(* CODESYS project BaseHts.library
   Company: Vistaprint
   Version: 0.0.0.48
   Description: 0.0.0.48 - Add AutoMode to HRU
      
      0.0.0.47 - Some Bugs in DPJ fixed
      
      0.0.0.46 - BaseElements 0.0.1.18
      	Some Bugs in DPJ, JUN fixed
      
      0.0.0.45 - BaseElements 0.0.1.17
      	MTR/sta_RUN Bug fixed
      
      0.0.0.44 - New Libs BasePLC 0.3.4.8, BaseElements 0.0.1.16
      
      0.0.0.43 - DPJ reworked (Missed Shirt Problem)
      
      0.0.0.42 - MER - new parameter added
      	HFE reworked
      
      0.0.0.41 - BasePLC V0.3.4.5; BaseElements V0.0.1.9
      
      0.0.0.40 - Add MTR Parameter dinWaitBetweenSensorAndReservation_um
      
      0.0.0.39 - Bug fixed in HFE, CHD; FOC and FOD added
      
      0.0.0.34 - JUN / DPJ replaced with version from Shirtstream
      
      0.0.0.32 - HFE from Lvl1 to Lvl2 and reworked
      
      0.0.0.30 - BaseElements 0.0.1.5 BasePLC 0.3.4.3 included, Tc2_SerialCom
      
      0.0.0.29 - BaseElements 0.0.1.2 BasePLC 0.3.4.2 included; FB_CtrlModule moved to BaseElements
      
      0.0.0.28 - Added ADS data channel to FB_HPS
      for shirt request from Heatpress
      
      0.0.0.27 - Added bolStopReleaseHangers
      
      0.0.0.26 - DPJ.sta_RUN Entry action reworked
      
      0.0.0.25 - Error JUN changed
      
      0.0.0.24 - Rising Edge detection of bolBringShirt in HPS
      
      0.0.0.23 - HTS, hanger turned line wait at SEP
      
      0.0.0.22 - Bug fixed in STOPbusy
      
      0.0.0.21 - Bugs fixed in HPS
      
      0.0.0.20 - HPS with new Child SEP
      	New BaseElements 0.0.0.20
      
      0.0.0.19 - Alternativ status for run sequence added; Timing reworked in MER jam detection;
      DPJ STOPBusy reworked, HRU Errors reworked, DPJ new Errors 12 and 13 added
      
      0.0.0.18 - Timeout Run / Stop sequence added
      
      0.0.0.17 - EMO reworked in BaseCtrlModule; CHD "destination full" reworked; AddStpGrp, AddRunGrp removed
      
      0.0.0.16 - Back to BasePLC Lib. V3.3.5 beacuase of PageFaults
      
      0.0.0.15 - Rebuild
      
      0.0.0.14 - Bugzilla ID 03: BufferFull for LineControl added
      
      0.0.0.13 - Bugzilla ID 55: reworked refill of SLB/STB
      
      0.0.0.12 - Update of BasePLC 0.3.3.7, BaseElements 0.0.0.17
      
      0.0.0.11 - Add more controllers to the library (LAI, CHD, HFE, PLS, JUN, DPJ, MER, HRU, HPS, COS, STB, SLB)
      
      0.0.0.10 - Clear pending command to prevent automatic recovery in sta_STOPBusy
      
      0.0.0.9 - BugFix in sub state "cSTA_SUB_CHECK_GROUP_STATUS" from run and stop sequence. Insert new "bolChecked" flag to detect if the sequence has been processed correctly.
      
      0.0.0.8 - Add TSTOP in checkChildAlmClass
      
      0.0.0.7- General revision of behaviour in case of emergency off (state EOFF) and general error (state ERROR). New handling for module specific interface.
      
      0.0.0.6 - Go to EOFFBusy if not in sta_EOFF
      
      0.0.0.5 - In Always: go to EOFFBusy at generalFault
      
      0.0.0.4 - In Always: go to EOFFBusy not to EOFF at emergency stop
      
      0.0.0.3 - Remove CurrentItemCounter and his inputs
      
      0.0.0.2 - Changes after first use in simulation in ICL Module
      
      0.0.0.1 - First release
   Author: AVME/DSC
   Title: Base_Hts

Project tree, tasks and I/O mapping:
  libraries: Base_Elements, 0.0.1.18 (Vistaprint); Base_PLC, 0.3.4.8 (Vistaprint); Tc2_Standard, 3.3.0.0 (Beckhoff Automation GmbH); Tc2_System, 3.3.5.0 (Beckhoff Automation GmbH); Tc2_Utilities, 3.3.7.0 (Beckhoff Automation GmbH); Tc3_Module, 3.3.5.0 (Beckhoff Automation GmbH)
  POUs/
    Controller/
      Driver/
        FOD/
          Infrastructure/
            function block FB_DecodeCanRxMessage [ST]
            function block fb_GenerateCanTxMessage [ST]
          function block FB_ReceiveFolderState [ST]: init
          function block FB_SendFolderMessage [ST]: init
          data type T_FOD
          data type T_FOD_Cfg
          data type T_FOD_Cur
          data type T_FOD_StateMachine
      Lvl0/
        CHD (Cross Hanger Detection)/
          global variables CHD_CmdState
          global variables Const_CHD
          function block FB_CHD [ST]: Always, FB_init, getCmdState, getCtrlSIf, IoInBridge, IoOutBridge, sta_ERROR, sta_ERRORQuit, sta_OFF, sta_OFFBusy, sta_PON, sta_RUN, sta_RUNBusy, sta_STOP, sta_STOPBusy, StateMachine
          data type T_CheckElement
          data type T_Ctrl_SIf_CHD
          data type T_Ctrl_SIf_CHD_Cfg
          data type T_Ctrl_SIf_CHD_Cur
          data type T_Ctrl_SIf_CHD_In
          data type T_Ctrl_SIf_CHD_Out
          data type T_Ctrl_SIf_CHD_Par
        FOC (Folder Communication)/
          function block FB_FOC [ST]: Always, FB_init, getCmdState, getCtrlSIf, IoInBridge, IoOutBridge, sta_ERROR, sta_OFF, sta_RELEASE, sta_RUN, sta_RUNbusy, StateMachine
          global variables FOC_CmdState
          data type T_Ctrl_SIf_FOC
          data type T_Ctrl_SIf_FOC_Cfg
          data type T_Ctrl_SIf_FOC_Cur
          data type T_Ctrl_SIf_FOC_In
          data type T_Ctrl_SIf_FOC_Out
          data type T_Ctrl_SIf_FOC_Par
        HRU (Hanger Rotation Unit)/
          function block FB_HRU [ST]: Always, FB_init, getCmdState, getCtrlSIf, IoInBridge, IoOutBridge, sta_EJECT, sta_EJECTBusy, sta_OFF, sta_OFFBusy, sta_RETRACT, sta_RETRACTBusy, sta_ROTATE, sta_ROTATEBusy, sta_RUN, sta_RUNBusy, sta_STOP, sta_STOPBusy, StateMachine
          global variables HRU_CmdState
          data type T_Ctrl_SIf_HRU
          data type T_Ctrl_SIf_HRU_In
          data type T_Ctrl_SIf_HRU_Out
          data type T_Ctrl_SIf_HRU_Par
        JUN (Junction)/
          data type E_Typ_JUN
          function block FB_JUN [ST]: Always, FB_init, getCmdState, getCtrlSIf, IoInBridge, IoOutBridge, sta_ERROR, sta_ERRORQuit, sta_OFF, sta_OFFBusy, sta_PON, sta_RELEASE, sta_RELEASE_ALL, sta_RELEASE_ALLBusy, sta_RELEASEBusy, sta_RUN, sta_RUNBusy, sta_STOP, sta_STOPBusy, StateMachine
          global variables JUN_CmdState
          data type T_Ctrl_SIf_JUN
          data type T_Ctrl_SIf_JUN_Cfg
          data type T_Ctrl_SIf_JUN_Cur
          data type T_Ctrl_SIf_JUN_Ilk
          data type T_Ctrl_SIf_JUN_In
          data type T_Ctrl_SIf_JUN_Out
          data type T_Ctrl_SIf_JUN_Par
          data type T_JUN_OutfeedCheck
        LAI (Labler Interface)/
          function block FB_LAI [ST]: Always, FB_init, getCmdState, getCtrlSIf, IoInBridge, IoOutBridge, sta_ERROR, sta_OFF, sta_OFFBusy, sta_RUN, sta_RUNBusy, StateMachine
          data type T_Ctrl_SIf_LAI
          data type T_Ctrl_SIf_LAI_Cfg
          data type T_Ctrl_SIf_LAI_Cur
          data type T_Ctrl_SIf_LAI_In
          data type T_Ctrl_SIf_LAI_Out
          data type T_Ctrl_SIf_LAI_Par
        PLS (PickToLight System)/
          global variables Const_PLS
          function block FB_PLS [ST]: Always, CtrlInit, FB_init, getCmdState, getCtrlSIf, IoInBridge, IoOutBridge, sta_ERROR, sta_ERRORQuit, sta_OFF, sta_RUN, StateMachine
          data type T_Ctrl_SIf_PLS
          data type T_Ctrl_SIf_PLS_Cfg
          data type T_Ctrl_SIf_PLS_Cur
          data type T_Ctrl_SIf_PLS_In
          data type T_Ctrl_SIf_PLS_Out
          data type T_Ctrl_SIf_PLS_Par
        STB (Stopper buffer)/
          function block FB_STB [ST]: Always, BufferFull, FB_init, getCmdState, getCtrlSIf, IoInBridge, IoOutBridge, MaxCapacity, NumOfHangers, sta_ERROR, sta_OFF, sta_OFFBusy, sta_RELEASE, sta_RELEASE_ALL, sta_RELEASE_ALLBusy, sta_RELEASEBusy, sta_RUN, sta_RUNBusy, sta_STOP, sta_STOPBusy, StateMachine
          global variables STB_CmdState
          data type T_Ctrl_SIf_STB
          data type T_Ctrl_SIf_STB_Cfg
          data type T_Ctrl_SIf_STB_Cur
          data type T_Ctrl_SIf_STB_Ilk
          data type T_Ctrl_SIf_STB_In
          data type T_Ctrl_SIf_STB_Out
          data type T_Ctrl_SIf_STB_Par
      Lvl1/
        DPJ (DecisionPoint Junction)/
          global variables Const_DPJ
          global variables DPJ_CmdState
          data type E_Decision_Job
          data type E_DecisionState
          data type E_ProductFlowState
          function block FB_DPJ [ST]: AddJunction, Always, checkAlmClassAllMultiChild, checkChildAlmClass, checkChildPointer, checkStateAllMultiChild, CmdToAllMultiChild, CtrlInit, DtChnToPLC_Decision, FB_init, getCtrlSIf, IoInBridge, IoOutBridge, SetAlmClassAllMultiChild, sta_ERROR, sta_ERRORQuit, sta_OFF, sta_OFFBusy, sta_PON, sta_RUN, sta_RUNBusy, sta_STOP, sta_STOPBusy, StateMachine
          function block FB_DtChnToLine_JobDone [ST]: Creat
          data type T_Ctrl_SIf_DPJ
          data type T_Ctrl_SIf_DPJ_Cfg
          data type T_Ctrl_SIf_DPJ_Cur
          data type T_Ctrl_SIf_DPJ_DtChnToLine
          data type T_Ctrl_SIf_DPJ_DtChnToPLC
          data type T_Ctrl_SIf_DPJ_In
          data type T_Ctrl_SIf_DPJ_Out
          data type T_Ctrl_SIf_DPJ_Par
          data type T_Decision
          data type T_Decision_DtChn
          data type T_DecisionElement
          data type T_JobDone_DtChn
          data type T_SimDtChn
        SLB (Slide buffer)/
          global variables Const_SLB
          function block FB_SLB [ST]: AddBufferZone, Always, BufferFull, CalcMaxCapacity, CalcSumNumOfHangers, checkAllZonesEmpty, checkAllZonesFull, checkChildAlmClass, checkChildValid, checkStateAllZones, CmdToAllZones, CtrlInit, FB_init, getCmdState, getCtrlSIf, IoInBridge, IoOutBridge, MaxCapacity, NumOfHangers, RefillZones, RefillZones_parallel, sta_OFF, sta_RELEASE_ALL, sta_RELEASE_ALLBusy, sta_RUN, sta_RUNBusy, sta_STOP, sta_STOPBusy, StateMachine
          global variables SLB_CmdState
          data type T_Ctrl_SIf_SLB
          data type T_Ctrl_SIf_SLB_Cfg
          data type T_Ctrl_SIf_SLB_Cur
          data type T_Ctrl_SIf_SLB_In
          data type T_Ctrl_SIf_SLB_Par
      Lvl2/
        COS (Control Station)/
          global variables COS_CmdState
          function block FB_COS [ST]: Always, checkChildAlmClass, CtrlInit, FB_init, getCmdState, getCtrlSIf, IoInBridge, sta_OFF, sta_RUN, sta_RUNBusy, sta_STOP, sta_STOPBusy, StateMachine
          data type T_Ctrl_SIf_COS
          data type T_Ctrl_SIf_COS_Cfg
          data type T_Ctrl_SIf_COS_Cur
          data type T_Ctrl_SIf_COS_In
          data type T_Ctrl_SIf_COS_Par
        FOL (Folder)/
          function block FB_FOL [ST]: Always, checkChildAlmClass, CtrlInit, FB_init, getCmdState, getCtrlSIf, IoInBridge, IoOutBridge, sta_OFF, sta_RUN, sta_RUNBusy, StateMachine
          global variables FOL_CmdState
          data type T_Ctrl_SIf_FOL
          data type T_Ctrl_SIf_FOL_Cfg
          data type T_Ctrl_SIf_FOL_Cur
          data type T_Ctrl_SIf_FOL_In
          data type T_Ctrl_SIf_FOL_Out
          data type T_Ctrl_SIf_FOL_Par
        HFE/
          global variables Const_HFE
          function block FB_HFE [ST]: AddJunction, Always, checkChildPointer, CtrlInit, FB_init, getCtrlSIf, IoInBridge, IoOutBridge, Refill, sta_OFF, sta_RUN, sta_RUNBusy, StateMachine
          data type T_Ctrl_SIf_HFE
          data type T_Ctrl_SIf_HFE_Cfg
          data type T_Ctrl_SIf_HFE_Cur
          data type T_Ctrl_SIf_HFE_Par
        HPS (Heat Press Shirt Station)/
          global variables Const_HPS
          data type E_DtChnJob
          function block FB_DtChnToLine_ChargeDone [ST]: Creat
          function block FB_HPS [ST]: AddDrive, Always, checkChildAlmClass, checkChildPointer, checkStateAllMultiChild, CmdToAllMultiChild, CtrlInit, DtChnToPLC_NewCharge, FB_init, getCmdState, getCtrlSIf, IoInBridge, IoOutBridge, RefillTurnedLine, sta_OFF, sta_RUN, sta_RUNBusy, sta_STOP, sta_STOPBusy, StateMachine
          data type T_ChargeDone_DtChn
          data type T_Ctrl_SIf_HPS
          data type T_Ctrl_SIf_HPS_Ads
          data type T_Ctrl_SIf_HPS_Ads_Read
          data type T_Ctrl_SIf_HPS_Cfg
          data type T_Ctrl_SIf_HPS_Cur
          data type T_Ctrl_SIf_HPS_DtChnToLine
          data type T_Ctrl_SIf_HPS_DtChnToPLC
          data type T_Ctrl_SIf_HPS_In
          data type T_Ctrl_SIf_HPS_Out
          data type T_Ctrl_SIf_HPS_Par
          data type T_NewCharge_DtChn
        MER (Merger Standard)/
          global variables Const_MER
          data type E_Typ_MER_AUTO_MODE
          data type E_Typ_MER_MODE
          function block FB_MER [ST]: AddLine, Always, BufferFull, CalcMaxCapacity, CalcSumOfItems, checkChildAlmClass, checkChildValid, checkStateAllLines, CmdToAllLines, CtrlInit, FB_init, getCmdState, getCtrlSIf, IoInBridge, IoOutBridge, MaxCapacity, NumOfHangers, sta_OFF, sta_RUN, sta_RUNBusy, sta_STOP, sta_STOPBusy, StateMachine
          data type T_Ctrl_SIf_MER
          data type T_Ctrl_SIf_MER_Cfg
          data type T_Ctrl_SIf_MER_Cur
          data type T_Ctrl_SIf_MER_In
          data type T_Ctrl_SIf_MER_Par
          data type T_Line
        MTR (Merger Transport)/
          global variables Const_MTR
          data type E_Typ_MTR_SECTION_STATE
          function block FB_MTR [ST]: AddLine, Always, BufferFull, CalcMaxCapacity, CalcSumOfItems, checkChildAlmClass, checkChildValid, checkStateAllLines, CmdToAllLines, CtrlInit, FB_init, getCtrlSIf, IoInBridge, MaxCapacity, NumOfHangers, sta_OFF, sta_RUN, sta_RUNBusy, sta_STOP, sta_STOPBusy, StateMachine
          data type T_Ctrl_SIf_MTR
          data type T_Ctrl_SIf_MTR_Cfg
          data type T_Ctrl_SIf_MTR_Cur
          data type T_Ctrl_SIf_MTR_In
          data type T_Ctrl_SIf_MTR_Par
          data type T_MTR_Buffer_Sections
      Lvl3/
    Utility Functions/
  Version/
    global variables Global_Version
*)

// POUs/Controller/Driver/FOD/T_FOD
TYPE T_FOD :
STRUCT
	strState: STRING;
	strCmd: STRING;
	intCmd: INT;
	intServiceCmd: INT;
	stStatus: T_RFD_Status;
	Cfg: T_FOD_Cfg;
	Cur: T_FOD_Cur;
END_STRUCT
END_TYPE

// POUs/Controller/Driver/FOD/T_FOD_Cfg
TYPE T_FOD_Cfg :
STRUCT
END_STRUCT
END_TYPE

// POUs/Controller/Driver/FOD/T_FOD_Cur
TYPE T_FOD_Cur :
STRUCT
END_STRUCT
END_TYPE

// POUs/Controller/Driver/FOD/T_FOD_StateMachine
TYPE T_FOD_StateMachine :
STRUCT
	///actual state
	intState: INT;
	///state of last cycle
	intStateLastCycle: INT;
	///save history backup p.e. in ERROR state
	intStateHistory: INT;
	///set state for next cycle
	intStateNext: INT;
	///Time in this State
	udiTimeInState_ms: UDINT;
END_STRUCT
END_TYPE

// POUs/Controller/Lvl0/CHD (Cross Hanger Detection)/T_CheckElement
TYPE T_CheckElement :
STRUCT
	eState: E_DecisionState;
	dinActPos_um: DINT;
END_STRUCT
END_TYPE

// POUs/Controller/Lvl0/CHD (Cross Hanger Detection)/T_Ctrl_SIf_CHD
TYPE T_Ctrl_SIf_CHD :
STRUCT
	///configuration
	Cfg: T_Ctrl_SIf_CHD_Cfg;
	///parameter
	Par: T_Ctrl_SIf_CHD_Par;
	///current values
	Cur: T_Ctrl_SIf_CHD_Cur;
	///io input
	In: T_Ctrl_SIf_CHD_In;
	///io output
	Out: T_Ctrl_SIf_CHD_Out;
	///alarm number used in this controller
	Alm: ARRAY[1..4] OF T_Ctrl_Alm;
END_STRUCT
END_TYPE

// POUs/Controller/Lvl0/CHD (Cross Hanger Detection)/T_Ctrl_SIf_CHD_Cfg
TYPE T_Ctrl_SIf_CHD_Cfg :
STRUCT
	/// Option called "Schiefe Bügel"
	bolHasInconsistentHangerSensor: BOOL;
	/// Option called "Leerbügelerkennung"
	bolHasEmptyHangerSensor: BOOL;
	/// Option
	bolHasSlideFullSensor: BOOL;
	/// Option
	bolStopAtRejact: BOOL;
END_STRUCT
END_TYPE

// POUs/Controller/Lvl0/CHD (Cross Hanger Detection)/T_Ctrl_SIf_CHD_Cur
TYPE T_Ctrl_SIf_CHD_Cur :
STRUCT
	///[um] actual position from the transport written from Parent
	dinTransportPosition_um: DINT;
	///[um] actual speed from the transport written from Parent
	dinTransportspeed_um_s: DINT;
	///[um] actual calculated position
	dinTransportPositionCalc_um: DINT;
	/// junction is open
	bolOpen: BOOL;
	///sensor hanger passed
	bolPassed: BOOL;
	///counter double hanger
	udintCounterDoubleHanger: UDINT;
END_STRUCT
END_TYPE

// POUs/Controller/Lvl0/CHD (Cross Hanger Detection)/T_Ctrl_SIf_CHD_In
TYPE T_Ctrl_SIf_CHD_In :
STRUCT
	/// Sensor hanger passed the junction	
	bolPassed: T_Ctrl_IoBool;
	/// Sensor double hanger
	bolSensorDoubleHanger: T_Ctrl_IoBoolDebounced;
	/// Sensor inconsistent hanger (as option)
	bolSensorInconsistentHanger: T_Ctrl_IoBool;
	/// Sensor empty hanger (as option)
	bolSensorEmptyHanger: T_Ctrl_IoBool;
	/// Button (as option)
	bolButtonRestartTLP: T_Ctrl_IoBool;
END_STRUCT
END_TYPE

// POUs/Controller/Lvl0/CHD (Cross Hanger Detection)/T_Ctrl_SIf_CHD_Out
TYPE T_Ctrl_SIf_CHD_Out :
STRUCT
	///switch valve junction
	bolOpen: T_Ctrl_IoBool;
	/// Blow light sensor
	bolBlow: T_Ctrl_IoBool;
	/// Info light (as option)
	bolLightTLPStopedByCHD: T_Ctrl_IoBool;
END_STRUCT
END_TYPE

// POUs/Controller/Lvl0/CHD (Cross Hanger Detection)/T_Ctrl_SIf_CHD_Par
TYPE T_Ctrl_SIf_CHD_Par :
STRUCT
	///[ms] until junction is open
	udiOpenTime_ms: UDINT;
	///[ms] until junction is closed
	udiCloseTime_ms: UDINT;
	///[ms] until failure timeout passing sensor is set?
	udiPassTime_ms: UDINT;
	///[ms] simulation time for passing the stopper or /2 of timeout time?
	udiSimPassTime_ms: UDINT;
	/// [um] Position of the junction
	dinPosition_um: DINT;
	/// [um] Distance from open to close position
	dinOpenWay_um: DINT;
	/// [um] Distance from first to last sensor
	dinDistanceBetweenSensors_DoubleHangerFirst_um: DINT;
	/// [um] Distance from first to last sensor
	dinDistanceBetweenSensors_EmptyHangerFirst_um: DINT;
	/// [um] PinDistance
	dinPinDistance_um: DINT;
	/// [ms] Time until jam at slide detected
	udinTimeUntilJam_ms: UDINT;
	/// [ms] Valve open time
	udiPulseLengthBlowValve_ms: UDINT;
	/// [ms] Valve closed time
	udiIntervalLengthBlowValve_ms: UDINT;
	/// [ms] Debounce time until double hanger sends cross-hanger-detected-signal. Prevents jitter.
	udiDebounceTimeDoubleHanger_ms: UDINT;
END_STRUCT
END_TYPE

// POUs/Controller/Lvl0/FOC (Folder Communication)/T_Ctrl_SIf_FOC
TYPE T_Ctrl_SIf_FOC :
STRUCT
	///configuration
	Cfg: T_Ctrl_SIf_FOC_Cfg;
	///parameter
	Par: T_Ctrl_SIf_FOC_Par;
	///current values
	Cur: T_Ctrl_SIf_FOC_Cur;
	///io input
	In: T_Ctrl_SIf_FOC_In;
	///io output
	Out: T_Ctrl_SIf_FOC_Out;
	///alarm number used in this controller
	Alm: ARRAY[1..5] OF T_Ctrl_Alm;
END_STRUCT
END_TYPE

// POUs/Controller/Lvl0/FOC (Folder Communication)/T_Ctrl_SIf_FOC_Cfg
TYPE T_Ctrl_SIf_FOC_Cfg :
STRUCT
	/// CAN identifier of sender (thats us)
	intCobId: INT;
	/// CAN identifier of receiver (Folder)
	intFolderCobId: INT;
	/// [ms] Given CAN msg command from LineControl. When no DataReadReady signal it's an error!
	udiMissingDataReadReadyTimeout_ms: UDINT;
	/// [ms] Given DataReadReady signal. When LineControl sends no CAN msg command it's an error!
	udiMissingCanMsgTimeout_ms: UDINT;
END_STRUCT
END_TYPE

// POUs/Controller/Lvl0/FOC (Folder Communication)/T_Ctrl_SIf_FOC_Cur
TYPE T_Ctrl_SIf_FOC_Cur :
STRUCT
	/// filtered data read ready counter
	uliDataReadReadyCounter: ULINT;
	/// filtered empty hanger counter
	uliEmptyHangerCounter: ULINT;
	/// overall number of sent CAN messages to folder
	uliCountSentMessages: ULINT;
	/// counter for warnings when DataReadReady window was detected but no RFID CAN cmd was sent by LineControl. This means shirt stack of 1 as fallback.
	uliWarningsDataReadReadyButNoRfid: ULINT;
END_STRUCT
END_TYPE

// POUs/Controller/Lvl0/FOC (Folder Communication)/T_Ctrl_SIf_FOC_In
TYPE T_Ctrl_SIf_FOC_In :
STRUCT
	usiCANDeviceErrorState: T_Ctrl_IoUsint;
END_STRUCT
END_TYPE

// POUs/Controller/Lvl0/FOC (Folder Communication)/T_Ctrl_SIf_FOC_Out
TYPE T_Ctrl_SIf_FOC_Out :
STRUCT
END_STRUCT
END_TYPE

// POUs/Controller/Lvl0/FOC (Folder Communication)/T_Ctrl_SIf_FOC_Par
TYPE T_Ctrl_SIf_FOC_Par :
STRUCT
	/// number of messages to send cyclic after an event (for redundancy)
	intNumberOfSendMessages: INT;
	/// filter receiving CAN messages for DataReadReady and EmptyHangerOnTheWay to prevent jitters
	tFilterTimeCanMessages: TIME;
	/// [ms] Duration of sending release CAN messages to Folder. This time will be also used for clearing the CAN flag again.
	udiTimeReleaseCanMessage_ms: UDINT;
	/// [ms] Waiting time before RELEASE_SHIRTS is possible. To ensure tact stop, last folded shirt must be on the stack.
	udiWaitTimeBeforeRelease_ms: UDINT;
END_STRUCT
END_TYPE

// POUs/Controller/Lvl0/HRU (Hanger Rotation Unit)/T_Ctrl_SIf_HRU
TYPE T_Ctrl_SIf_HRU :
STRUCT
	///configuration
	///parameter
	Par: T_Ctrl_SIf_HRU_Par;
	///current values
	///io input
	In: T_Ctrl_SIf_HRU_In;
	///io output
	Out: T_Ctrl_SIf_HRU_Out;
	///alarm number used in this controller
	Alm: ARRAY[1..4] OF T_Ctrl_Alm;
END_STRUCT
END_TYPE

// POUs/Controller/Lvl0/HRU (Hanger Rotation Unit)/T_Ctrl_SIf_HRU_In
TYPE T_Ctrl_SIf_HRU_In :
STRUCT
	///sensor hanger in rotation unit
	bolHangerDetected: T_Ctrl_IoBool;
END_STRUCT
END_TYPE

// POUs/Controller/Lvl0/HRU (Hanger Rotation Unit)/T_Ctrl_SIf_HRU_Out
TYPE T_Ctrl_SIf_HRU_Out :
STRUCT
	/// Valve Rotate hanger 180°
	bolRotate: T_Ctrl_IoBool;
	/// Valve eject hanger
	bolEject: T_Ctrl_IoBool;
END_STRUCT
END_TYPE

// POUs/Controller/Lvl0/HRU (Hanger Rotation Unit)/T_Ctrl_SIf_HRU_Par
TYPE T_Ctrl_SIf_HRU_Par :
STRUCT
	///[ms] time for eject (no sensor exist)
	udiEjectTime_ms: UDINT;
	///[ms] time for retract (no sensor exist)
	udiRetractTime_ms: UDINT;
	///[ms] time for rotate (no sensor exist)
	udiRotateTime_ms: UDINT;
	///[ms] wait time with hanger at sensor for start rotating
	udiWaitForRotate_ms: UDINT;
	///[ms] simulate the next hanger
	udiSimNextHangerTime_ms: UDINT;
	/// [ms] Timeout to detect a hanger in the rotation unit
	udiTimeOutHRU_Hanger_ms: UDINT;
	/// Enable AutoMode, used for example at the RotaryHeatPress Output
	bolAutoModeEnable: BOOL;
END_STRUCT
END_TYPE

// POUs/Controller/Lvl0/JUN (Junction)/E_Typ_JUN
TYPE E_Typ_JUN :
(
	Max_E_Typ_JUN
);
END_TYPE

// POUs/Controller/Lvl0/JUN (Junction)/T_Ctrl_SIf_JUN
TYPE T_Ctrl_SIf_JUN :
STRUCT
	///configuration
	Cfg: T_Ctrl_SIf_JUN_Cfg;
	///parameter
	Par: T_Ctrl_SIf_JUN_Par;
	///current values
	Cur: T_Ctrl_SIf_JUN_Cur;
	///io input
	In: T_Ctrl_SIf_JUN_In;
	///io output
	Out: T_Ctrl_SIf_JUN_Out;
	///alarm number used in this controller
	Alm: ARRAY[1..4] OF T_Ctrl_Alm;
	///interlock of output/movements
	Ilk: T_Ctrl_SIf_JUN_Ilk;
END_STRUCT
END_TYPE

// POUs/Controller/Lvl0/JUN (Junction)/T_Ctrl_SIf_JUN_Cfg
TYPE T_Ctrl_SIf_JUN_Cfg :
STRUCT
	eTyp: E_Typ_JUN;
	/// Number of the target
	dinTargetNr: DINT;
END_STRUCT
END_TYPE

// POUs/Controller/Lvl0/JUN (Junction)/T_Ctrl_SIf_JUN_Cur
TYPE T_Ctrl_SIf_JUN_Cur :
STRUCT
	///[um] actual position from the transport written from Parent
	dinTransportPosition_um: DINT;
	///[um] actual speed from the transport written from Parent
	dinTransportspeed_um_s: DINT;
	///[um] actual calculated position
	dinTransportPositionCalc_um: DINT;
	/// junction is open
	bolOpen: BOOL;
	///sensor hanger passed
	bolPassed: BOOL;
END_STRUCT
END_TYPE

// POUs/Controller/Lvl0/JUN (Junction)/T_Ctrl_SIf_JUN_Ilk
TYPE T_Ctrl_SIf_JUN_Ilk :
STRUCT
	///interlock Open the junction 
	bolOpen: BOOL;
END_STRUCT
END_TYPE

// POUs/Controller/Lvl0/JUN (Junction)/T_Ctrl_SIf_JUN_In
TYPE T_Ctrl_SIf_JUN_In :
STRUCT
	///sensor hanger passed the junction
	bolPassed: Base_PLC.T_Ctrl_IoBoolDebounced;
END_STRUCT
END_TYPE

// POUs/Controller/Lvl0/JUN (Junction)/T_Ctrl_SIf_JUN_Out
TYPE T_Ctrl_SIf_JUN_Out :
STRUCT
	///switch valve retract
	bolOpen: T_Ctrl_IoBool;
END_STRUCT
END_TYPE

// POUs/Controller/Lvl0/JUN (Junction)/T_Ctrl_SIf_JUN_Par
TYPE T_Ctrl_SIf_JUN_Par :
STRUCT
	///[ms] until junction is open
	udiOpenTime_ms: UDINT;
	///[ms] until junction is closed
	udiCloseTime_ms: UDINT;
	///[ms] until failure timeout passing sensor is set?
	udiPassTime_ms: UDINT;
	///[ms] simulation time for passing the stopper or /2 of timeout time?
	udiSimPassTime_ms: UDINT;
	/// Position of the junction
	dinPosition_um: DINT;
	/// Distance from open to close position
	dinOpenWay_um: DINT;
	/// Pointer to Hashtable from Desicion
	pTblDecision: POINTER TO ARRAY[0..cintMaxDecisions] OF T_DecisionElement;
	/// [ms] Debounce time until passed hanger sends signal. Prevents jitter.
	udiDebounceTimePassed_ms: UDINT;
END_STRUCT
END_TYPE

// POUs/Controller/Lvl0/JUN (Junction)/T_JUN_OutfeedCheck
TYPE T_JUN_OutfeedCheck :
STRUCT
	/// Time for check
	udiTime_ms: UDINT;
	/// Index of the Hashtable
	intHTIndex: INT;
END_STRUCT
END_TYPE

// POUs/Controller/Lvl0/LAI (Labler Interface)/T_Ctrl_SIf_LAI
TYPE T_Ctrl_SIf_LAI :
STRUCT
	///configuration
	Cfg: T_Ctrl_SIf_LAI_Cfg;
	///parameter
	Par: T_Ctrl_SIf_LAI_Par;
	///current values
	Cur: T_Ctrl_SIf_LAI_Cur;
	///io input
	In: T_Ctrl_SIf_LAI_In;
	///io output
	Out: T_Ctrl_SIf_LAI_Out;
	///alarm number used in this controller
	Alm: ARRAY[1..7] OF T_Ctrl_Alm;
END_STRUCT
END_TYPE

// POUs/Controller/Lvl0/LAI (Labler Interface)/T_Ctrl_SIf_LAI_Cfg
TYPE T_Ctrl_SIf_LAI_Cfg :
STRUCT
END_STRUCT
END_TYPE

// POUs/Controller/Lvl0/LAI (Labler Interface)/T_Ctrl_SIf_LAI_Cur
TYPE T_Ctrl_SIf_LAI_Cur :
STRUCT
	/// Signal from Labler Job finished
	bolJobFinished: BOOL;
END_STRUCT
END_TYPE

// POUs/Controller/Lvl0/LAI (Labler Interface)/T_Ctrl_SIf_LAI_In
TYPE T_Ctrl_SIf_LAI_In :
STRUCT
	bolReady: T_Ctrl_IoBool;
	bolNoError: T_Ctrl_IoBool;
	bolLowMaterial: T_Ctrl_IoBool;
	bolJobFinished: T_Ctrl_IoBool;
	bolCylInPosition: T_Ctrl_IoBool;
	bolErrLabel: T_Ctrl_IoBool;
	bolErrPrinter: T_Ctrl_IoBool;
	bolErrDrive: T_Ctrl_IoBool;
	bolErrCylinder: T_Ctrl_IoBool;
END_STRUCT
END_TYPE

// POUs/Controller/Lvl0/LAI (Labler Interface)/T_Ctrl_SIf_LAI_Out
TYPE T_Ctrl_SIf_LAI_Out :
STRUCT
	bolAutomaticOn: T_Ctrl_IoBool;
	bolProductInPos: T_Ctrl_IoBool;
END_STRUCT
END_TYPE

// POUs/Controller/Lvl0/LAI (Labler Interface)/T_Ctrl_SIf_LAI_Par
TYPE T_Ctrl_SIf_LAI_Par :
STRUCT
	/// [ms] Timeout supervision ready signal
	udi_TimeoutReady_ms: UDINT;
	/// [ms] Simulation of Ready signal
	udi_SimReady_ms: UDINT;
	/// [ms] Simulation of pulse finished signal
	udi_Finished_ms: UDINT;
END_STRUCT
END_TYPE

// POUs/Controller/Lvl0/PLS (PickToLight System)/T_Ctrl_SIf_PLS
TYPE T_Ctrl_SIf_PLS :
STRUCT
	///configuration
	///parameter
	///current values
	Cur: T_Ctrl_SIf_PLS_Cur;
	///io input
	In: T_Ctrl_SIf_PLS_In;
	///io output
	Out: T_Ctrl_SIf_PLS_Out;
	///alarm number used in this controller
	Alm: ARRAY[1..6] OF T_Ctrl_Alm;
END_STRUCT
END_TYPE

// POUs/Controller/Lvl0/PLS (PickToLight System)/T_Ctrl_SIf_PLS_Cfg
TYPE T_Ctrl_SIf_PLS_Cfg :
STRUCT
END_STRUCT
END_TYPE

// POUs/Controller/Lvl0/PLS (PickToLight System)/T_Ctrl_SIf_PLS_Cur
TYPE T_Ctrl_SIf_PLS_Cur :
STRUCT
	dinCounter: DINT;
END_STRUCT
END_TYPE

// POUs/Controller/Lvl0/PLS (PickToLight System)/T_Ctrl_SIf_PLS_In
TYPE T_Ctrl_SIf_PLS_In :
STRUCT
END_STRUCT
END_TYPE

// POUs/Controller/Lvl0/PLS (PickToLight System)/T_Ctrl_SIf_PLS_Out
TYPE T_Ctrl_SIf_PLS_Out :
STRUCT
END_STRUCT
END_TYPE

// POUs/Controller/Lvl0/PLS (PickToLight System)/T_Ctrl_SIf_PLS_Par
TYPE T_Ctrl_SIf_PLS_Par :
STRUCT
END_STRUCT
END_TYPE

// POUs/Controller/Lvl0/STB (Stopper buffer)/T_Ctrl_SIf_STB
TYPE T_Ctrl_SIf_STB :
STRUCT
	/// configuration
	Cfg: T_Ctrl_SIf_STB_Cfg;
	/// parameter
	Par: T_Ctrl_SIf_STB_Par;
	/// current values
	Cur: T_Ctrl_SIf_STB_Cur;
	/// io input
	In: T_Ctrl_SIf_STB_In;
	/// io output
	Out: T_Ctrl_SIf_STB_Out;
	/// alarm number used in this controller
	Alm: ARRAY[1..4] OF T_Ctrl_Alm;
	/// interlock of output/movements
	Ilk: T_Ctrl_SIf_STB_Ilk;
END_STRUCT
END_TYPE

// POUs/Controller/Lvl0/STB (Stopper buffer)/T_Ctrl_SIf_STB_Cfg
TYPE T_Ctrl_SIf_STB_Cfg :
STRUCT
	/// Has buffer full sensor (optional)
	bolHasBufferFullSensor: BOOL;
	/// Has hanger detection sensor
	bolHasHangerDetection: BOOL;
	/// Has decrement sensor, if not then decrement with stroke 
	bolHasDecrementSensor: BOOL;
	/// Don't delete dinNumOfHangersInBuffer if no hanger detected, used for very long buffers
	bolDisableBufferDelete: BOOL;
	/// Max. buffer capacity
	dinMaxCapacity: DINT;
	/// Number of passing hangers per pulse
	uinNumOfHangersPerPulse: UINT;
	/// max number of hangers detected in STOP if bolCylPosLostMonitoring activated until an error occures
	dinMaxNumOfHangers_PosMonitoring: DINT;
	/// Enable cylinder position lost monitoring
	bolCylPosLostMonitoring: BOOL;
	/// to release all work with puleses and counts or use time to release
	bolReleaseAllNonPulse: BOOL;
	/// Unique line number. (Starts with 1..) Used in case if STB work in combination with FUB MTR to merge hangers into a TLK.
	usiLineNumber: USINT;
	/// Simulation mode
	/// 0 = Normal simulation of STB function, e.g. STB in combination with SLB controller
	/// 1 = Hanger detection signal can be overridden manually to test STB in combination with MTR controller
	usiSimulationMode: USINT;
END_STRUCT
END_TYPE

// POUs/Controller/Lvl0/STB (Stopper buffer)/T_Ctrl_SIf_STB_Cur
TYPE T_Ctrl_SIf_STB_Cur :
STRUCT
	/// Hangers passed total counter (reset in state OFF)
	dinHangersPassedTotal: DINT;
	/// Hangers passed package counter (is updated when “RELEASE_ALL” command is completed)
	dinHangersPassedPackage: DINT;
	/// Hanger detected
	bolHangerDetected: BOOL;
	/// Approximate number of hangers in buffer
	dinNumOfHangersInBuffer: DINT;
	/// Buffer is full
	bolBufferFull: BOOL;
	/// Pointer to section buffer of FUB MTR. Needed in case if STB work in combination with MTR to merge hangers into a TLK.
	pSectionBuffer: POINTER TO ARRAY[0..Const_MTR.cusiSectionBuffer_SIZE] OF T_MTR_Buffer_Sections;
	///[um] actual position from the transport written from Parent
	dinTransportPosition_um: DINT;
	///[um] actual speed from the transport written from Parent
	dinTransportspeed_um_s: DINT;
	///[um] actual calculated position
	dinTransportPositionCalc_um: DINT;
END_STRUCT
END_TYPE

// POUs/Controller/Lvl0/STB (Stopper buffer)/T_Ctrl_SIf_STB_Ilk
TYPE T_Ctrl_SIf_STB_Ilk :
STRUCT
	/// interlock retraction of cylinder
	bolRetract: BOOL;
END_STRUCT
END_TYPE

// POUs/Controller/Lvl0/STB (Stopper buffer)/T_Ctrl_SIf_STB_In
TYPE T_Ctrl_SIf_STB_In :
STRUCT
	/// Sensor hanger detected
	bolHangerDetected: T_Ctrl_IoBoolDebounced;
	/// Sensor buffer full
	bolBufferFull: T_Ctrl_IoBoolDebounced;
	/// Sensor decrement counter (option)
	bolDecrementCounter: T_Ctrl_IoBoolDebounced;
END_STRUCT
END_TYPE

// POUs/Controller/Lvl0/STB (Stopper buffer)/T_Ctrl_SIf_STB_Out
TYPE T_Ctrl_SIf_STB_Out :
STRUCT
	/// Output for controlling the pneumatic cylinder 
	/// if bolRetract2 is not used  = 1 -> second pin up first pin (inlet) down second up 
	bolRetract: T_Ctrl_IoBool;
	/// = 1 -> second pin down (outlet)
	bolRetract2: T_Ctrl_IoBool;
END_STRUCT
END_TYPE

// POUs/Controller/Lvl0/STB (Stopper buffer)/T_Ctrl_SIf_STB_Par
TYPE T_Ctrl_SIf_STB_Par :
STRUCT
	/// [ms] Pulse length valve (clocking)
	udiPulseLengthValve_ms: UDINT;
	/// [ms] Interval buffer emptying
	udiIntervalBufferEmptying_ms: UDINT;
	/// [ms] Timeout buffer emptying (0 = disable monitoring)
	udiTimeoutBufferEmptying_ms: UDINT;
	/// [ms] Timedelay sensor signal valid
	udiSensorTime_ms: UDINT;
	/// Buffermode: 0= Emptying buffer, use buffer capacity at cycle start
	///             1= Emptying buffer, newly added hangers will be considered
	usiBuffermode: USINT;
	/// [ms] Time for release all hangers
	udiReleaseAllTime_ms: UDINT;
	/// [ms] Debounce time for inputs
	udiDebounceTime_ms: UDINT;
	/// This parameter is used in combination with FB_MTR
	/// [um] Position of the end of slide (must be measured, starts at pin sensor [zero pos], ends at the point where the slide comes in the transport)
	dinPositionOfSlide_um: DINT;
	/// This parameter is used in combination with FB_MTR	
	/// [ms] Time on slide.
	uinTimeOnSlide_ms: UINT;
END_STRUCT
END_TYPE

// POUs/Controller/Lvl1/DPJ (DecisionPoint Junction)/E_Decision_Job
TYPE E_Decision_Job :
(
	none := 0,
	NEW := 1,
	REPLACE_ID := 2,
	DELETE_ID := 3,
	DELETE_JUNCTION := 4,
	DELETE_ALL := 5,
	MAX_E_Decision_Job
);
END_TYPE

// POUs/Controller/Lvl1/DPJ (DecisionPoint Junction)/E_DecisionState
TYPE E_DecisionState :
(
	none := 0,
	Wait := 1,
	WayToJunction := 2,
	OnJunction := 3,
	Processed := 4,
	DriveOut := 5,
	Finished := 6,
	MAX_E_DecisionState
);
END_TYPE

// POUs/Controller/Lvl1/DPJ (DecisionPoint Junction)/E_ProductFlowState
TYPE E_ProductFlowState :
(
	none := 0,
	busy,
	done,
	error
);
END_TYPE

// POUs/Controller/Lvl1/DPJ (DecisionPoint Junction)/T_Ctrl_SIf_DPJ
TYPE T_Ctrl_SIf_DPJ :
STRUCT
	///configuration
	Cfg: T_Ctrl_SIf_DPJ_Cfg;
	///parameter
	Par: T_Ctrl_SIf_DPJ_Par;
	///current values
	Cur: T_Ctrl_SIf_DPJ_Cur;
	///io input
	In: T_Ctrl_SIf_DPJ_In;
	///io output
	///Data Channel from Line Controller to PLC
	DtChnToPLC: T_Ctrl_SIf_DPJ_DtChnToPLC;
	///Data Channel from PLC to Line Controller
	DtChnToLine: T_Ctrl_SIf_DPJ_DtChnToLine;
	///alarm number used in this controller
	Alm: ARRAY[1..15] OF T_Ctrl_Alm;
END_STRUCT
END_TYPE

// POUs/Controller/Lvl1/DPJ (DecisionPoint Junction)/T_Ctrl_SIf_DPJ_Cfg
TYPE T_Ctrl_SIf_DPJ_Cfg :
STRUCT
	eTyp: E_Typ_JUN;
	/// Maximale buffer capacity
	dinMaxCapacity: DINT;
	/// Number of junctions
	intCountJunctions: INT;
	/// Decisionpoint has a Hangerdetection sensor for exactly position reading
	bolHangerDetectionExist: BOOL;
	/// Send every Done Job to Line controller
	bolDtChToLine_send: BOOL;
	/// Simulation of the Speed internal, do not read Pos and speed from Transport
	bolSimSpeedInternal: BOOL;
	/// Stop when Hanger passed the last instead of selected junction, else just Info
	bolStopAtPassLastJunction: BOOL;
	/// Number of elements in aTblDecision
	intMaxDecisions: INT;
	/// Simulate line control data channels
	bolSimDtChLine: BOOL;
	bolSimEnableDtChToPLC: BOOL;
END_STRUCT
END_TYPE

// POUs/Controller/Lvl1/DPJ (DecisionPoint Junction)/T_Ctrl_SIf_DPJ_Cur
TYPE T_Ctrl_SIf_DPJ_Cur :
STRUCT
	///[um] actual position from the transport written from Parent
	dinTransportPosition_um: DINT;
	///[um] actual speed from the transport written from Parent
	dinTransportspeed_um_s: DINT;
	///Max capacity calculated from all childs 
	dinMaxCapacity: DINT;
	///Actual Item Count of this controller with all childs
	dinCurrentItemCount: DINT;
	/// Childs output is ready, written by Parent
	a_bolJunctionOutputOK: ARRAY[0..Base_Const.cMaxNrOfChilds] OF BOOL;
	/// [um] Distance to the farthest (last) junction, determined in "CtrlInit" 
	dinDistanceToFarthestJunction: DINT;
END_STRUCT
END_TYPE

// POUs/Controller/Lvl1/DPJ (DecisionPoint Junction)/T_Ctrl_SIf_DPJ_DtChnToLine
TYPE T_Ctrl_SIf_DPJ_DtChnToLine :
STRUCT
	stJobDone: T_JobDone_DtChn;
END_STRUCT
END_TYPE

// POUs/Controller/Lvl1/DPJ (DecisionPoint Junction)/T_Ctrl_SIf_DPJ_DtChnToPLC
TYPE T_Ctrl_SIf_DPJ_DtChnToPLC :
STRUCT
	stNewDecision: T_Decision_DtChn;
END_STRUCT
END_TYPE

// POUs/Controller/Lvl1/DPJ (DecisionPoint Junction)/T_Ctrl_SIf_DPJ_In
TYPE T_Ctrl_SIf_DPJ_In :
STRUCT
	bolHangerDetector: T_Ctrl_IoBool;
	bolCounterIn: T_Ctrl_IoBool;
	bolCounterOut: T_Ctrl_IoBool;
END_STRUCT
END_TYPE

// POUs/Controller/Lvl1/DPJ (DecisionPoint Junction)/T_Ctrl_SIf_DPJ_Out
TYPE T_Ctrl_SIf_DPJ_Out :
STRUCT
	///switch valve retract
	bolRetract: T_Ctrl_IoBool;
	///switch valve extend
	bolExtend: T_Ctrl_IoBool;
END_STRUCT
END_TYPE

// POUs/Controller/Lvl1/DPJ (DecisionPoint Junction)/T_Ctrl_SIf_DPJ_Par
TYPE T_Ctrl_SIf_DPJ_Par :
STRUCT
	/// Timeout communication at Datachannel
	udiTimeOutRead_ms: UDINT;
	/// Maximal time until delete a Job
	udiTimeMaxJob_s: UDINT;
	/// [um] Offset to distance of the farthest junction. 
	/// Defines the point, where a job will be automatically deleted from the buffer, if destination junction was not defined.  
	dinDistanceOffsetUntilDelJob_um: DINT;
	dinSimTimeAcknowledgeDataChl_ms: DINT;
	dinSimProcessTimeOnLineCtrl_ms: DINT;
	dinSimTarget: DINT;
	intSimDischargingEveryXtenHanger: INT;
	// Timeout time for waiting for the second signal (Sensor or RFID) 
	udiWaitingForSecondSignalTimeout_ms: UDINT;
END_STRUCT
END_TYPE

// POUs/Controller/Lvl1/DPJ (DecisionPoint Junction)/T_Decision
TYPE T_Decision :
STRUCT
	strID: STRING(16);
	uliRFID: ULINT;
	/// junction nr.
	dinTarget: DINT;
END_STRUCT
END_TYPE

// POUs/Controller/Lvl1/DPJ (DecisionPoint Junction)/T_Decision_DtChn
TYPE T_Decision_DtChn :
STRUCT
	stDecision: T_Decision;
	intJob: INT;
	intDataState: INT;
END_STRUCT
END_TYPE

// POUs/Controller/Lvl1/DPJ (DecisionPoint Junction)/T_DecisionElement
TYPE T_DecisionElement :
STRUCT
	stDecision: T_Decision;
	dtTimeJob: DT;
	dtTimeRFID: DT;
	eState: E_DecisionState;
	dinActPos_um: DINT;
END_STRUCT
END_TYPE

// POUs/Controller/Lvl1/DPJ (DecisionPoint Junction)/T_JobDone_DtChn
TYPE T_JobDone_DtChn :
STRUCT
	stDecision: T_Decision;
	strTimestamp: STRING(24);
	intDataState: INT;
END_STRUCT
END_TYPE

// POUs/Controller/Lvl1/DPJ (DecisionPoint Junction)/T_SimDtChn
TYPE T_SimDtChn :
STRUCT
	stDecision: T_Decision;
	intJob: INT;
	strTimestamp: STRING(24);
	intDataState: INT;
	/// 0=undef, 1=SimDataPLCToLineDone, 2=SimDataLineToPLCInWork
	intInternalSimState: USINT;
END_STRUCT
END_TYPE

// POUs/Controller/Lvl1/SLB (Slide buffer)/T_Ctrl_SIf_SLB
TYPE T_Ctrl_SIf_SLB :
STRUCT
	/// configuration
	Cfg: T_Ctrl_SIf_SLB_Cfg;
	/// parameter
	Par: T_Ctrl_SIf_SLB_Par;
	/// current values
	Cur: T_Ctrl_SIf_SLB_Cur;
	/// io input
	In: T_Ctrl_SIf_SLB_In;
	/// io output
	/// ...no physical Output
	/// alarm number used in this controller
	Alm: ARRAY[1..3] OF T_Ctrl_Alm;
END_STRUCT
END_TYPE

// POUs/Controller/Lvl1/SLB (Slide buffer)/T_Ctrl_SIf_SLB_Cfg
TYPE T_Ctrl_SIf_SLB_Cfg :
STRUCT
	// Enable Refill parallel (For example in HFE used)
	bolRefill_parallel: BOOL;
END_STRUCT
END_TYPE

// POUs/Controller/Lvl1/SLB (Slide buffer)/T_Ctrl_SIf_SLB_Cur
TYPE T_Ctrl_SIf_SLB_Cur :
STRUCT
	/// Number of buffer zones, depends on how many times the method "AddBufferZone" was called at init
	usiNumOfBufferZones: USINT;
	/// Hanger detected -> based on zone 1, output
	bolHangerDetected: BOOL;
	/// Hangers passed total counter -> based on zone 1, output (reset in state OFF)
	dinHangersPassedTotal: DINT;
	/// Hangers passed package counter -> based on zone 1, output (is updated when “RELEASE_ALL” command is completed)
	dinHangersPassedPackage: DINT;
	/// Approximate number of hangers in buffer -> based on all zones
	dinNumOfHangersInBuffer: DINT;
	/// Max. buffer capacity -> based on all zones
	dinMaxCapacity: DINT;
	/// Input buffer is full -> based on last zone full signal
	bolInputBufferFull: BOOL;
	/// All buffers full -> based on all zones
	bolAllBuffersFull: BOOL;
	/// Number of passing hangers per pulse in first zone
	uinNumOfHangersPerPulseFirstZone: UINT;
END_STRUCT
END_TYPE

// POUs/Controller/Lvl1/SLB (Slide buffer)/T_Ctrl_SIf_SLB_In
TYPE T_Ctrl_SIf_SLB_In :
STRUCT
END_STRUCT
END_TYPE

// POUs/Controller/Lvl1/SLB (Slide buffer)/T_Ctrl_SIf_SLB_Par
TYPE T_Ctrl_SIf_SLB_Par :
STRUCT
	/// [ms] Interval buffer emptying
	udiIntervalBufferEmptying_ms: UDINT;
	/// [ms] Interval buffer filling
	udiIntervalBufferFilling_ms: UDINT;
	///[ms] simulation time for hanger coming in
	udiSimIncomingTime_ms: UDINT;
END_STRUCT
END_TYPE

// POUs/Controller/Lvl2/COS (Control Station)/T_Ctrl_SIf_COS
TYPE T_Ctrl_SIf_COS :
STRUCT
	///configuration
	Cfg: T_Ctrl_SIf_COS_Cfg;
	///parameter
	Par: T_Ctrl_SIf_COS_Par;
	///current values
	Cur: T_Ctrl_SIf_COS_Cur;
	///io input
	In: T_Ctrl_SIf_COS_In;
	///alarm number used in this controller
	Alm: ARRAY[1..8] OF T_Ctrl_Alm;
END_STRUCT
END_TYPE

// POUs/Controller/Lvl2/COS (Control Station)/T_Ctrl_SIf_COS_Cfg
TYPE T_Ctrl_SIf_COS_Cfg :
STRUCT
END_STRUCT
END_TYPE

// POUs/Controller/Lvl2/COS (Control Station)/T_Ctrl_SIf_COS_Cur
TYPE T_Ctrl_SIf_COS_Cur :
STRUCT
END_STRUCT
END_TYPE

// POUs/Controller/Lvl2/COS (Control Station)/T_Ctrl_SIf_COS_In
TYPE T_Ctrl_SIf_COS_In :
STRUCT
	bolNextShirt: T_Ctrl_IoBool;
END_STRUCT
END_TYPE

// POUs/Controller/Lvl2/COS (Control Station)/T_Ctrl_SIf_COS_Par
TYPE T_Ctrl_SIf_COS_Par :
STRUCT
END_STRUCT
END_TYPE

// POUs/Controller/Lvl2/FOL (Folder)/T_Ctrl_SIf_FOL
TYPE T_Ctrl_SIf_FOL :
STRUCT
	///configuration
	Cfg: T_Ctrl_SIf_FOL_Cfg;
	///parameter
	Par: T_Ctrl_SIf_FOL_Par;
	///current values
	Cur: T_Ctrl_SIf_FOL_Cur;
	///io input
	In: T_Ctrl_SIf_FOL_In;
	///io output
	Out: T_Ctrl_SIf_FOL_Out;
	///alarm number used in this controller
	Alm: ARRAY[1..6] OF T_Ctrl_Alm;
END_STRUCT
END_TYPE

// POUs/Controller/Lvl2/FOL (Folder)/T_Ctrl_SIf_FOL_Cfg
TYPE T_Ctrl_SIf_FOL_Cfg :
STRUCT
END_STRUCT
END_TYPE

// POUs/Controller/Lvl2/FOL (Folder)/T_Ctrl_SIf_FOL_Cur
TYPE T_Ctrl_SIf_FOL_Cur :
STRUCT
	/// overall item counter
	dinMaxCapacity: DINT;
	bolIsFull: BOOL;
END_STRUCT
END_TYPE

// POUs/Controller/Lvl2/FOL (Folder)/T_Ctrl_SIf_FOL_In
TYPE T_Ctrl_SIf_FOL_In :
STRUCT
END_STRUCT
END_TYPE

// POUs/Controller/Lvl2/FOL (Folder)/T_Ctrl_SIf_FOL_Out
TYPE T_Ctrl_SIf_FOL_Out :
STRUCT
END_STRUCT
END_TYPE

// POUs/Controller/Lvl2/FOL (Folder)/T_Ctrl_SIf_FOL_Par
TYPE T_Ctrl_SIf_FOL_Par :
STRUCT
	///udiHangerLoadingTime_ms	: UDINT;	// time delay for clamping and for separator to bring a hanger into LST chain
	udiTimeNextHangers_ms: UDINT;
END_STRUCT
END_TYPE

// POUs/Controller/Lvl2/HFE/T_Ctrl_SIf_HFE
TYPE T_Ctrl_SIf_HFE :
STRUCT
	///configuration
	Cfg: T_Ctrl_SIf_HFE_Cfg;
	///parameter
	Par: T_Ctrl_SIf_HFE_Par;
	///current values
	Cur: T_Ctrl_SIf_HFE_Cur;
	///alarm number used in this controller
	Alm: ARRAY[1..6] OF T_Ctrl_Alm;
END_STRUCT
END_TYPE

// POUs/Controller/Lvl2/HFE/T_Ctrl_SIf_HFE_Cfg
TYPE T_Ctrl_SIf_HFE_Cfg :
STRUCT
	/// Number of supportetd LDS
	uintNbOfLDS: UINT;
END_STRUCT
END_TYPE

// POUs/Controller/Lvl2/HFE/T_Ctrl_SIf_HFE_Cur
TYPE T_Ctrl_SIf_HFE_Cur :
STRUCT
END_STRUCT
END_TYPE

// POUs/Controller/Lvl2/HFE/T_Ctrl_SIf_HFE_Par
TYPE T_Ctrl_SIf_HFE_Par :
STRUCT
	// Waiting between SLB-STB Close and Junction open
	udiWaitingTime_ms: UDINT;
	// Open junction time
	a_udiTimeOpen_ms: ARRAY[0..cuintMaxStation] OF UDINT;
	// Close junction time
	a_udiTimeClose_ms: ARRAY[0..cuintMaxStation] OF UDINT;
	// Enable Junction to LDS
	a_bolEnableJunction: ARRAY[0..cuintMaxStation] OF BOOL;
END_STRUCT
END_TYPE

// POUs/Controller/Lvl2/HPS (Heat Press Shirt Station)/E_DtChnJob
TYPE E_DtChnJob :
(
	none := 0,
	NEW := 1,
	REPLACE_ID := 2,
	DELETE_ID := 3,
	DELETE_JUNCTION := 4,
	DELETE_ALL := 5,
	MAX_E_Decision_Job
);
END_TYPE

// POUs/Controller/Lvl2/HPS (Heat Press Shirt Station)/T_ChargeDone_DtChn
TYPE T_ChargeDone_DtChn :
STRUCT
	intLine: INT;
	dtTimestamp: DT;
	intDataState: INT;
END_STRUCT
END_TYPE

// POUs/Controller/Lvl2/HPS (Heat Press Shirt Station)/T_Ctrl_SIf_HPS
TYPE T_Ctrl_SIf_HPS :
STRUCT
	///configuration
	Cfg: T_Ctrl_SIf_HPS_Cfg;
	///parameter
	Par: T_Ctrl_SIf_HPS_Par;
	///current values
	Cur: T_Ctrl_SIf_HPS_Cur;
	///io input
	In: T_Ctrl_SIf_HPS_In;
	///io output
	Out: T_Ctrl_SIf_HPS_Out;
	///ADS data channel from heatpress
	Ads: T_Ctrl_SIf_HPS_Ads;
	///Data Channel from Line Controller to PLC
	DtChnToPLC: T_Ctrl_SIf_HPS_DtChnToPLC;
	///Data Channel from PLC to Line Controller
	DtChnToLine: T_Ctrl_SIf_HPS_DtChnToLine;
	///alarm number used in this controller
	Alm: ARRAY[1..9] OF T_Ctrl_Alm;
END_STRUCT
END_TYPE

// POUs/Controller/Lvl2/HPS (Heat Press Shirt Station)/T_Ctrl_SIf_HPS_Ads
TYPE T_Ctrl_SIf_HPS_Ads :
STRUCT
	stRead		: T_Ctrl_SIf_HPS_Ads_Read;
END_STRUCT
END_TYPE

// POUs/Controller/Lvl2/HPS (Heat Press Shirt Station)/T_Ctrl_SIf_HPS_Ads_Read
TYPE T_Ctrl_SIf_HPS_Ads_Read :
STRUCT
	// Request for front shirt send from Heatpress 
	udiRequestFrontShirt: 		UDINT;
	// Request for back shirt send from Heatpress
	udiRequestBackShirt: 		UDINT;
END_STRUCT
END_TYPE

// POUs/Controller/Lvl2/HPS (Heat Press Shirt Station)/T_Ctrl_SIf_HPS_Cfg
TYPE T_Ctrl_SIf_HPS_Cfg :
STRUCT
	/// Maximale buffer capacity only this controller without childs
	dinMaxCapacity: DINT;
	/// Send every Done Job to Line controller
	bolDtChToLine_send: BOOL;
END_STRUCT
END_TYPE

// POUs/Controller/Lvl2/HPS (Heat Press Shirt Station)/T_Ctrl_SIf_HPS_Cur
TYPE T_Ctrl_SIf_HPS_Cur :
STRUCT
	///Max capacity calculated from all childs 
	dinMaxCapacity: DINT;
	///Actual Item Count of this controller with all childs
	dinCurrentItemCount: DINT;
END_STRUCT
END_TYPE

// POUs/Controller/Lvl2/HPS (Heat Press Shirt Station)/T_Ctrl_SIf_HPS_DtChnToLine
TYPE T_Ctrl_SIf_HPS_DtChnToLine :
STRUCT
	stChargeDone: T_ChargeDone_DtChn;
END_STRUCT
END_TYPE

// POUs/Controller/Lvl2/HPS (Heat Press Shirt Station)/T_Ctrl_SIf_HPS_DtChnToPLC
TYPE T_Ctrl_SIf_HPS_DtChnToPLC :
STRUCT
	stNewCharge: T_NewCharge_DtChn;
END_STRUCT
END_TYPE

// POUs/Controller/Lvl2/HPS (Heat Press Shirt Station)/T_Ctrl_SIf_HPS_In
TYPE T_Ctrl_SIf_HPS_In :
STRUCT
	bolCounterIn1: T_Ctrl_IoBool;
	bolCounterIn2: T_Ctrl_IoBool;
	bolCounterOut1: T_Ctrl_IoBool;
	bolCounterOut2: T_Ctrl_IoBool;
	bolBringShirtStraight: T_Ctrl_IoBool;
	bolBringShirtTurned: T_Ctrl_IoBool;
END_STRUCT
END_TYPE

// POUs/Controller/Lvl2/HPS (Heat Press Shirt Station)/T_Ctrl_SIf_HPS_Out
TYPE T_Ctrl_SIf_HPS_Out :
STRUCT
	/// Interface to Heatpress without LineControl
	bolShirtStraightReady: T_Ctrl_IoBool;
	bolShirtTurnReady: T_Ctrl_IoBool;
END_STRUCT
END_TYPE

// POUs/Controller/Lvl2/HPS (Heat Press Shirt Station)/T_Ctrl_SIf_HPS_Par
TYPE T_Ctrl_SIf_HPS_Par :
STRUCT
	/// Timeout communication at Datachannel
	udiTimeOutRead_ms: UDINT;
	/// [ms] Time to wait for starting a new drive
	udiTimeDriveStart_ms: UDINT;
	/// [ms] Time to wait for stopping a new drive
	udiTimeDriveStop_ms: UDINT;
	/// [ms] Interval buffer filling
	udiIntervalBufferFilling_ms: UDINT;
END_STRUCT
END_TYPE

// POUs/Controller/Lvl2/HPS (Heat Press Shirt Station)/T_NewCharge_DtChn
TYPE T_NewCharge_DtChn :
STRUCT
	intLine: INT;
	intJob: INT;
	intDataState: INT;
END_STRUCT
END_TYPE

// POUs/Controller/Lvl2/MER (Merger Standard)/E_Typ_MER_AUTO_MODE
TYPE E_Typ_MER_AUTO_MODE :
(
	/// 0= Merge over time 	
	MergeOverTime := 0,
	/// 1= Merge over setpoint (number of hangers)
	MergeOverSetpoint
);
END_TYPE

// POUs/Controller/Lvl2/MER (Merger Standard)/E_Typ_MER_MODE
TYPE E_Typ_MER_MODE :
(
	/// 0= main mode automatic, controller automatically merge hangers from different lines dependent E_Typ_MER_AUTO_MODE
	Automatic := 0,
	/// 1= main mode on command, in case if merger work as charge controller. Release line X dependent from parent command.
	OnCommand
);
END_TYPE

// POUs/Controller/Lvl2/MER (Merger Standard)/T_Ctrl_SIf_MER
TYPE T_Ctrl_SIf_MER :
STRUCT
	/// configuration
	Cfg: T_Ctrl_SIf_MER_Cfg;
	/// parameter
	Par: T_Ctrl_SIf_MER_Par;
	/// current values
	Cur: T_Ctrl_SIf_MER_Cur;
	/// io input
	In: T_Ctrl_SIf_MER_In;
	/// io output
	/// ...no physical Output
	/// alarm number used in this controller
	Alm: ARRAY[1..3] OF T_Ctrl_Alm;
END_STRUCT
END_TYPE

// POUs/Controller/Lvl2/MER (Merger Standard)/T_Ctrl_SIf_MER_Cfg
TYPE T_Ctrl_SIf_MER_Cfg :
STRUCT
	/// Merger main mode
	usiMergeMainMode: E_Typ_MER_MODE;
	/// Number of jam sensors (option)
	usiCountJamSensors: USINT;
END_STRUCT
END_TYPE

// POUs/Controller/Lvl2/MER (Merger Standard)/T_Ctrl_SIf_MER_Cur
TYPE T_Ctrl_SIf_MER_Cur :
STRUCT
	/// Number of lines to merge, depends on how many times the method "AddLine" was called at init
	usiNumOfLinesToMerge: USINT;
	/// Approximate number of merged hangers total from all lines
	dinNumOfMergedHangersTotal: DINT;
	/// Max. buffer capacity -> based on all lines
	dinMaxCapacity: DINT;
	/// Actual Item Count of this controller -> based on all lines
	dinCurrentItemCount: DINT;
	/// Childs is ready
	a_bolChildReady: ARRAY[0..Base_Const.cMaxNrOfChilds] OF BOOL;
END_STRUCT
END_TYPE

// POUs/Controller/Lvl2/MER (Merger Standard)/T_Ctrl_SIf_MER_In
TYPE T_Ctrl_SIf_MER_In :
STRUCT
	/// Sensors for jam detection (option)
	a_bolJamSensor: ARRAY[1..cMAX_JAM_SENSORS] OF BASE_PLC.T_Ctrl_IoBool;
END_STRUCT
END_TYPE

// POUs/Controller/Lvl2/MER (Merger Standard)/T_Ctrl_SIf_MER_Par
TYPE T_Ctrl_SIf_MER_Par :
STRUCT
	/// Setpoint, line number to release all from parent in case if main mode "OnCommand" is selected. (1 -> X)
	usiLineNumToReleaseAll: USINT;
	/// List of parameters for Line 1 -> X
	a_LinePar: ARRAY[0..Base_Const.cMaxNrOfChilds] OF T_Line;
	/// [ms] Timeout jam sensor in RUN
	udi_jamTimeout_ms: UDINT;
	// Enable Release in Auto Mode, if a hanger exists
	a_bolEnableHangerRelease: ARRAY[0..Base_Const.cMaxNrOfChilds] OF BOOL;
END_STRUCT
END_TYPE

// POUs/Controller/Lvl2/MER (Merger Standard)/T_Line
TYPE T_Line :
STRUCT
	/// Merge-mode
	usiMergeMode: E_Typ_MER_AUTO_MODE;
	/// [ms] Time, how long hangers are merged from sub- into the main line.
	udiMergingTime_ms: UDINT;
	/// Setpoint, how many hangers should merged from sub- into the main line.
	uinNumOfHangersToMerge: UINT;
	/// [ms] Wait time until the line is free before release the next line to prevent hanger collision.
	udiWaitTimeLineFree_ms: UDINT;
END_STRUCT
END_TYPE

// POUs/Controller/Lvl2/MTR (Merger Transport)/E_Typ_MTR_SECTION_STATE
TYPE E_Typ_MTR_SECTION_STATE :
(
	/// 0 = Undefined (free buffer element) 
	Undefined := 0,
	/// 1 = section start position was set
	StartPositionSet := 1,
	/// 2 = section end position was set (section is free)
	EndPositionSet := 2,
	/// 3 = section already engaged, detected by hanger sensor. (hanger in section, set if hanger was detected by sensor) 
	EngagedByDetecSensor := 3,
	/// 4 = section reserved for line
	Reserved := 4,
	/// 5 = hanger on slide
	HangerOnSlide := 5,
	/// 6 = hanger was released in section from slide
	HangerReleased := 6
) USINT;
END_TYPE

// POUs/Controller/Lvl2/MTR (Merger Transport)/T_Ctrl_SIf_MTR
TYPE T_Ctrl_SIf_MTR :
STRUCT
	/// configuration
	Cfg: T_Ctrl_SIf_MTR_Cfg;
	/// parameter
	Par: T_Ctrl_SIf_MTR_Par;
	/// current values
	Cur: T_Ctrl_SIf_MTR_Cur;
	/// io input
	In: T_Ctrl_SIf_MTR_In;
	/// io output
	/// ...no physical Output
	/// alarm number used in this controller
	Alm: ARRAY[1..3] OF T_Ctrl_Alm;
END_STRUCT
END_TYPE

// POUs/Controller/Lvl2/MTR (Merger Transport)/T_Ctrl_SIf_MTR_Cfg
TYPE T_Ctrl_SIf_MTR_Cfg :
STRUCT
END_STRUCT
END_TYPE

// POUs/Controller/Lvl2/MTR (Merger Transport)/T_Ctrl_SIf_MTR_Cur
TYPE T_Ctrl_SIf_MTR_Cur :
STRUCT
	/// Number of lines to merge, depends on how many times the method "AddLine" was called at init
	usiNumOfLinesToMerge: USINT;
	/// Approximate number of merged hangers total from all lines
	dinNumOfMergedHangersTotal: DINT;
	/// Max. buffer capacity -> based on all lines
	dinMaxCapacity: DINT;
	/// Actual Item Count of this controller -> based on all lines
	dinCurrentItemCount: DINT;
	/// Childs is ready
	a_bolChildReady: ARRAY[0..Base_Const.cMaxNrOfChilds] OF BOOL;
	///[um] actual position from the transport written from Parent
	dinTransportPosition_um: DINT;
	///[um] actual speed from the transport written from Parent
	dinTransportspeed_um_s: DINT;
	///[um] actual calculated position
	dinTransportPositionCalc_um: DINT;
END_STRUCT
END_TYPE

// POUs/Controller/Lvl2/MTR (Merger Transport)/T_Ctrl_SIf_MTR_In
TYPE T_Ctrl_SIf_MTR_In :
STRUCT
	/// Sensor hanger detected
	bolHangerDetected: T_Ctrl_IoBool;
	/// Sensor pin from new section is detected
	bolPinDetected: T_Ctrl_IoBool;
END_STRUCT
END_TYPE

// POUs/Controller/Lvl2/MTR (Merger Transport)/T_Ctrl_SIf_MTR_Par
TYPE T_Ctrl_SIf_MTR_Par :
STRUCT
	/// [um] Pin Lenght
	dinPinLenght_um: DINT;
	/// [um] Section Lenght
	dinSectionLenght_um: DINT;
	/// [um] Trigger start offset
	dinTrigStartOffset_um: DINT;
	/// [um] Trigger end offset
	dinTrigEndOffset_um: DINT;
	/// [um] Hanger Detection Sensor Position (measured from ZEROPOINT)
	dinHangerSensorPosition_um: DINT;
	// [um] Wait between Hanger Detection Sensor Position and Reservation
	dinWaitBetweenSensorAndReservation_um: DINT;
END_STRUCT
END_TYPE

// POUs/Controller/Lvl2/MTR (Merger Transport)/T_MTR_Buffer_Sections
TYPE T_MTR_Buffer_Sections :
STRUCT
	/// Start position of the section (triggered by pin sensor)
	dinSecStartPos: DINT;
	/// End position of the section (triggered by pin sensor)
	dinSecEndPos: DINT;
	/// Calculated trigger start position within the section
	dinTrigStartPos: DINT;
	/// Calculated trigger end position within the section
	dinTrigEndPos: DINT;
	/// Note: Trigger start and end position defines the position window to release a hanger
	enmState: E_Typ_MTR_SECTION_STATE;
	/// Info for which line number the section is reserved for
	usiReservedForLine: USINT;
END_STRUCT
END_TYPE

// POUs/Controller/Lvl0/CHD (Cross Hanger Detection)/CHD_CmdState
VAR_GLOBAL
END_VAR

// POUs/Controller/Lvl0/CHD (Cross Hanger Detection)/Const_CHD
VAR_GLOBAL CONSTANT
	cuintMaxIndex: UINT := 10;
END_VAR

// POUs/Controller/Lvl0/FOC (Folder Communication)/FOC_CmdState
VAR_GLOBAL CONSTANT
	///ctrl commands definitions
	///specific commands >200 - every command has to be a even number
	cCMD_RELEASE_SHIRTS: INT := 201;
	///ctrl specific states definitions
	cSTA_RELEASE_SHIRTS: INT := cCMD_RELEASE_SHIRTS;
END_VAR

// POUs/Controller/Lvl0/HRU (Hanger Rotation Unit)/HRU_CmdState
VAR_GLOBAL CONSTANT
	///ctrl commands definitions
	///specific commands >200 - every command has to be a even number
	cCMD_RETRACT: INT := 202;
	cCMD_EJECT: INT := 204;
	cCMD_ROTATE: INT := 206;
	///ctrl specific states definitions
	cSTA_RETRACTBusy: INT := 201;
	cSTA_RETRACT: INT := cCMD_RETRACT;
	cSTA_EJECTBusy: INT := 203;
	cSTA_EJECT: INT := cCMD_EJECT;
	cSTA_ROTATEBusy: INT := 205;
	cSTA_ROTATE: INT := cCMD_ROTATE;
END_VAR

// POUs/Controller/Lvl0/JUN (Junction)/JUN_CmdState
VAR_GLOBAL CONSTANT
	///ctrl commands definitions
	///specific commands >200 - every command has to be a even number
	cCMD_RELEASE_ALL: INT := 302;
	cCMD_RELEASE: INT := 304;
	///ctrl specific states definitions
	cSTA_RELEASE_ALLBusy: INT := 301;
	cSTA_RELEASE_ALL: INT := cCMD_RELEASE_ALL;
	cSTA_RELEASEBusy: INT := 303;
	cSTA_RELEASE: INT := cCMD_RELEASE;
END_VAR

// POUs/Controller/Lvl0/PLS (PickToLight System)/Const_PLS
VAR_GLOBAL CONSTANT
	MAX_SKUS : INT := 11;
END_VAR

// POUs/Controller/Lvl0/STB (Stopper buffer)/STB_CmdState
VAR_GLOBAL CONSTANT
	/// ctrl commands definitions
	/// specific commands >200 - every command has to be a even number
	cCMD_RELEASE: INT := 306;
	/// Empties the whole buffer dependent the selected buffer mode
	cCMD_RELEASE_ALL: INT := 308;
	/// ctrl specific states definitions
	cSTA_RELEASEBusy: INT := 305;
	cSTA_RELEASE: INT := cCMD_RELEASE;
	cSTA_RELEASE_ALLBusy: INT := 307;
	cSTA_RELEASE_ALL: INT := cCMD_RELEASE_ALL;
END_VAR

// POUs/Controller/Lvl1/DPJ (DecisionPoint Junction)/Const_DPJ
VAR_GLOBAL CONSTANT
	/// Reduced, was 300
	cintMaxDecisions: INT := 100;
END_VAR

// POUs/Controller/Lvl1/DPJ (DecisionPoint Junction)/DPJ_CmdState
VAR_GLOBAL CONSTANT
	///ctrl commands definitions
	///specific commands >200 - every command has to be a even number
	cCMD_CLEAR: INT := 202;
END_VAR

// POUs/Controller/Lvl1/SLB (Slide buffer)/Const_SLB
VAR_GLOBAL CONSTANT
	cusiMinAddedChilds: USINT := 1;
END_VAR

// POUs/Controller/Lvl1/SLB (Slide buffer)/SLB_CmdState
VAR_GLOBAL CONSTANT
	/// ctrl commands definitions
	/// specific commands >200 - every command has to be a even number
	cCMD_RELEASE: INT := 306;
	/// Empties all buffer zones
	cCMD_RELEASE_ALL: INT := 308;
	/// ctrl specific states definitions
	cSTA_RELEASE_ALLBusy: INT := 307;
	cSTA_RELEASE_ALL: INT := cCMD_RELEASE_ALL;
END_VAR

// POUs/Controller/Lvl2/COS (Control Station)/COS_CmdState
VAR_GLOBAL CONSTANT
	///ctrl commands definitions
	///specific commands >200 - every command has to be a even number
	cCMD_RELEASE: INT := 306;
	/// ctrl specific states definitions
	cSTA_RELEASEBusy: INT := 305;
	cSTA_RELEASE: INT := cCMD_RELEASE;
END_VAR

// POUs/Controller/Lvl2/FOL (Folder)/FOL_CmdState
VAR_GLOBAL CONSTANT
	/// ctrl commands definitions
	/// specific commands >200 - every command has to be a even number
	///...needs no specific commands 
	cSTA_READY: UINT := 201;
END_VAR

// POUs/Controller/Lvl2/HFE/Const_HFE
VAR_GLOBAL CONSTANT
	cuintMaxStation: UINT := 4;
END_VAR

// POUs/Controller/Lvl2/HPS (Heat Press Shirt Station)/Const_HPS
VAR_GLOBAL CONSTANT
	cintMaxCharge: INT := 10;
END_VAR

// POUs/Controller/Lvl2/MER (Merger Standard)/Const_MER
VAR_GLOBAL CONSTANT
	cusiMinAddedChilds: USINT := 1;
	cMAX_JAM_SENSORS: USINT := 3;
END_VAR

// POUs/Controller/Lvl2/MTR (Merger Transport)/Const_MTR
VAR_GLOBAL CONSTANT
	cusiMinAddedChilds: USINT := 1;
	/// Buffer prepared for 80 sections, means, with section length e.g. 0.49 m a TLK with max. length of 39 m 
	cusiSectionBuffer_SIZE: USINT := 80;
END_VAR

// Version/Global_Version
// This function has been automatically generated from the project information.
VAR_GLOBAL CONSTANT
	{attribute 'const_non_replaced'}
	stLibVersion_Base_Hts : ST_LibVersion := (iMajor := 0, iMinor := 0, iBuild := 0, iRevision := 48, sVersion := '0.0.0.48');
END_VAR

// POUs/Controller/Driver/FOD/Infrastructure/FB_DecodeCanRxMessage
FUNCTION_BLOCK FB_DecodeCanRxMessage
VAR_INPUT
	RxMessage: CANQUEUE;
END_VAR
VAR_OUTPUT
	CobId: UINT;
	BytesReceived: UINT;
	arrDataReceived: CANMESSAGE;
END_VAR

BytesReceived := SHR((SHL(RxMessage.CobId,12)),12);
Cobid := SHR(rxMessage.CobId,5);
arrDataReceived := RxMessage.data;

END_FUNCTION_BLOCK

// POUs/Controller/Driver/FOD/Infrastructure/fb_GenerateCanTxMessage
FUNCTION_BLOCK fb_GenerateCanTxMessage
VAR_INPUT
	CobId: UINT;
	BytesToSend: UINT;
	arrDataToSend: CANMESSAGE;
END_VAR
VAR_OUTPUT
	TxMessage: CANQUEUE;
END_VAR

TxMessage.CobId := (SHL(CobId,5)) + BytesToSend;
TxMessage.data := arrDataToSend;

END_FUNCTION_BLOCK

// POUs/Controller/Driver/FOD/FB_ReceiveFolderState
FUNCTION_BLOCK FB_ReceiveFolderState
VAR_INPUT
	InRxCounter AT %I*: UINT;
	InNoOfRxMessages AT %I*: UINT;
	RxMessages AT %I*: ARRAY[0..9] OF CANQUEUE;
	/// CAN Identifier to listen for
	intCobId: INT := 112;
	/// time until DataReadReady windows gets detected (both directions: true and false). Use this to prevent jitters on the CAN bus.
	tFilterTime: TIME := TIME#100ms;
END_VAR
VAR_OUTPUT
	OutRxCounter AT %Q*: UINT;
	CpuOnline: BOOL;
	EmptyHangerOnTheWay: BOOL;
	FilteredEmptyHangerOnTheWay: BOOL;
	HangerRequest: BOOL;
	RequestData: BOOL;
	DataReadReady: BOOL;
	FilteredDataReadReady: BOOL;
	ErrorMessage: UINT;
	StatusMessage: UINT;
	/// non filtered counter
	uliCountDataReadReady: ULINT;
	/// non filtered counter
	uliCountEmptyHanger: ULINT;
	/// number of read CobId's	
	uliReadCounter: ULINT;
END_VAR
VAR
	tDataReadReadyTrue: TON;
	tDataReadReadyFalse: TON;
	tEmptyHangerOnTheWayTrue: TON;
	tEmptyHangerOnTheWayFalse: TON;
	/// current state
	uinState: UINT;
	/// last read CobId
	uinLastRxCobId: UINT;
	ReceivedBytes: UINT;
	arrDataRecieved: CANMESSAGE;
	k: UINT;
	fbDecodeRxMessage: fb_DecodeCanRxMessage;
END_VAR
VAR CONSTANT
	cSTA_WAIT_MESSAGE: UINT := 10;
	cSTA_SEARCH_MESSAGE: UINT := 20;
	cSTA_PARSE_MESSAGE: UINT := 30;
END_VAR

(*__________________________________________________________________________________________________
¦	
¦	Vistaprint Schweiz GmbH
¦	CH - 8401 Winterthur
¦
¦	www.vistaprint.ch - info@vistaprint.ch
¦___________________________________________________________________________________________________

Function desription:
CAN communication to Kannegiesser folder to listening for CAN messages and parse Folder state.


History:
Version		Date			Author		Comment
---------------------------------------------------------------------------------------------------
0.00.1		28.09.2013		VP/RE		Start history
0.00.2		28.10.2013		VP/RE		Handle multiple messages, filter for Folder message
0.00.3		29.10.2013		VP/RE		Introduced state names
0.00.4		11.12.2013		VP/RE		Implemented FilteredDataReadReady to prevent jitters in CAN communication 

___________________________________________________________________________________________________*)


CASE uinState OF
	
cSTA_WAIT_MESSAGE: 	
	IF InRxCounter <> OutRxCounter THEN
		uinState := cSTA_SEARCH_MESSAGE;
	END_IF
	
cSTA_SEARCH_MESSAGE:	
	FOR k := 0 TO InNoOfRxMessages DO
		fbDecodeRxMessage(	RxMessage:= RxMessages[k],
  							CobId=>uinLastRxCobId ,
							BytesReceived=> ReceivedBytes,
							arrDataReceived=>arrDataRecieved );

		// filter Folder message
		IF (uinLastRxCobId = INT_TO_UINT(intCobId)) THEN
			uinState := cSTA_PARSE_MESSAGE;
			EXIT;
		END_IF
			
	END_FOR
	
	IF (uinState = cSTA_SEARCH_MESSAGE) THEN
		uinState := cSTA_WAIT_MESSAGE;
	END_IF
	
	OutRxCounter := OutRxCounter + 1;
	
cSTA_PARSE_MESSAGE:	
	uliReadCounter := uliReadCounter + 1;
	
	// parse data
	CpuOnline := arrDataRecieved[0].0;
	EmptyHangerOnTheWay := arrDataRecieved[1].1;
	HangerRequest := arrDataRecieved[1].0;
	RequestData := arrDataRecieved[1].5;

	ErrorMessage := USINT_TO_UINT(arrDataRecieved[5]);
	StatusMessage := ANY_TO_UINT(arrDataRecieved[6] + arrDataRecieved[7] * 256);
	
	// update counters
	IF DataReadReady = FALSE AND arrDataRecieved[1].6 THEN
		uliCountDataReadReady := uliCountDataReadReady + 1;
	END_IF

	DataReadReady := arrDataRecieved[1].6;
	
	IF EmptyHangerOnTheWay = FALSE AND arrDataRecieved[1].1 THEN
		uliCountEmptyHanger := uliCountEmptyHanger + 1;
	END_IF
	
	uinState := cSTA_WAIT_MESSAGE;
	
END_CASE


// filter DataReadReady window
tDataReadReadyTrue(IN:= DataReadReady = TRUE , PT:= tFilterTime);
tDataReadReadyFalse(IN:= DataReadReady = FALSE , PT:= tFilterTime);
IF (tDataReadReadyTrue.Q = TRUE) THEN
	FilteredDataReadReady := TRUE;
END_IF
IF (tDataReadReadyFalse.Q = TRUE) THEN
	FilteredDataReadReady := FALSE;
END_IF

// filter EmptyHangerOnTheWay
tEmptyHangerOnTheWayTrue(IN:= EmptyHangerOnTheWay = TRUE , PT:= tFilterTime);
tEmptyHangerOnTheWayFalse(IN:= EmptyHangerOnTheWay = FALSE , PT:= tFilterTime);
IF (tEmptyHangerOnTheWayTrue.Q = TRUE) THEN
	FilteredEmptyHangerOnTheWay := TRUE;
END_IF
IF (tEmptyHangerOnTheWayFalse.Q = TRUE) THEN
	FilteredEmptyHangerOnTheWay := FALSE;
END_IF

METHOD init
OutRxCounter := InRxCounter;
uinState := cSTA_WAIT_MESSAGE;
END_METHOD

END_FUNCTION_BLOCK

// POUs/Controller/Driver/FOD/FB_SendFolderMessage
FUNCTION_BLOCK FB_SendFolderMessage
VAR_INPUT
	InTxCounter AT %I*: UINT;
	CpuOnline: BOOL;
	EmptyHangerConveying: BOOL;
	ProgramNumber: BYTE := 1;
	/// 1=forward, 2=sideward
	ShirtStackConveyor: BYTE := 1;
	ChangeCustomer: BOOL;
	StopFolder: BOOL;
	ShotOutStacks: BOOL;
	/// CAN Identifier of receiver
	TxCobId: UINT := 113;
	/// true = starts sending a message. make sure all data fields are set before.
	bStartSend: BOOL;
	/// timeout after sent message before next message will be send
	tTimeout: TIME := TIME#50ms;
END_VAR
VAR_OUTPUT
	TxMessages AT %Q*: ARRAY[0..9] OF CANQUEUE;
	OutTxCounter AT %Q*: UINT;
	OutNoOfTxMessages AT %Q*: UINT := 1;
END_VAR
VAR
	uinState: UINT;
	BytesToSend: UINT := 8;
	arrDataToSend: CANMESSAGE;
	m: UINT;
	fbGenerateTxMessage: fb_GenerateCanTxMessage;
	uliCountSentMessages: ULINT;
	tWaitTimer: TON;
END_VAR
VAR CONSTANT
	cSTA_WAIT_SEND: UINT := 10;
	cSTA_SEND_MESSAGE: UINT := 20;
	cSTA_WAIT_SEND_COMPLETE: UINT := 30;
	cSTA_WAIT_BEFORE_SEND_NEXT: UINT := 40;
END_VAR

(*__________________________________________________________________________________________________
¦	
¦	Vistaprint Schweiz GmbH
¦	CH - 8401 Winterthur
¦
¦	www.vistaprint.ch - info@vistaprint.ch
¦___________________________________________________________________________________________________

Function desription:
CAN communication to Kannegiesser folder to send commands.


History:
Version		Date			Author		Comment
---------------------------------------------------------------------------------------------------
0.00.1		28.09.2013		VP/RE		Start history
0.00.2		29.10.2013		VP/RE		Introduced state names
0.00.3		11.12.2013		VP/RE		Implemented sleep timeout after sending a CAN message.
___________________________________________________________________________________________________*)


CASE uinState OF
	
cSTA_WAIT_SEND:	
	IF bStartSend THEN
		bStartSend:=FALSE;
		uinState := cSTA_SEND_MESSAGE;
	END_IF
	
cSTA_SEND_MESSAGE:	
	
	uliCountSentMessages := uliCountSentMessages + 1;

	FOR m := 0 TO OutNoOfTxMessages - 1 DO
		
		arrDataToSend[0].0 := CpuOnline;
		arrDataToSend[0].1 := EmptyHangerConveying;
		arrDataToSend[1].0 := ChangeCustomer;
		
		arrDataToSend[0].4 := ProgramNumber.0;
		arrDataToSend[0].5 := ProgramNumber.1;
		arrDataToSend[0].6 := ProgramNumber.2;
		arrDataToSend[0].7 := ProgramNumber.3;
		
		IF (ShirtStackConveyor = 1) THEN
			arrDataToSend[2].1 := 1;
			arrDataToSend[2].2 := 0;
		ELSIF (ShirtStackConveyor = 2) THEN
			arrDataToSend[2].1 := 0;
			arrDataToSend[2].2 := 1;
		ELSIF (ShirtStackConveyor = 0) THEN
			arrDataToSend[2].1 := 0;
			arrDataToSend[2].2 := 0;
		END_IF
		
		arrDataToSend[3].5 := StopFolder;
		arrDataToSend[3].6 := ShotOutStacks;

		fbGenerateTxMessage(CobId := TxCobId,
							BytesToSend := BytesToSend,
							arrDataToSend := arrDataToSend ,
							TxMessage => TxMessages[0] );
	END_FOR
	
	OutTxCounter := OutTxCounter + 1;
	uinState := cSTA_WAIT_SEND_COMPLETE;
	
cSTA_WAIT_SEND_COMPLETE:	
	IF OutTxCounter = InTxCounter THEN
		uinState := cSTA_WAIT_BEFORE_SEND_NEXT;
	END_IF

cSTA_WAIT_BEFORE_SEND_NEXT:
	IF (tWaitTimer.Q = TRUE) THEN
		uinState := cSTA_WAIT_SEND;
	END_IF
	
END_CASE

tWaitTimer(IN := uinState = cSTA_WAIT_BEFORE_SEND_NEXT, PT := tTimeout);

METHOD init
uinState := cSTA_WAIT_SEND;
END_METHOD

END_FUNCTION_BLOCK

// POUs/Controller/Lvl0/CHD (Cross Hanger Detection)/FB_CHD
FUNCTION_BLOCK FB_CHD EXTENDS FB_CtrlBase
VAR_INPUT
	/// Sensor Slide full
	In_bolPassed: BOOL;
	/// Sensor double hanger
	In_bolDoubleHanger: BOOL;
	/// Sensor inconsistent hanger (as option)
	In_bolInconsistentHanger: BOOL;
	/// Sensor empty hanger (as option)
	In_bolEmptyHanger: BOOL;
	/// Button (as option)
	In_bolRestartTLP: BOOL;
END_VAR
VAR_OUTPUT
	/// switch valve junction
	Out_bolOpen: BOOL;
	/// Blow light sensor
	Out_bolBlow: BOOL;
	/// Info light (as option)
	Out_bolLightTLPStopedByCHD: BOOL;
END_VAR
VAR
	/// Specific interface struct for public access
	SIf: T_Ctrl_SIf_CHD;
	/// standard Loop variable
	uinI: UINT;
	/// Index to next job in Hashtable
	uintNextHastableIdx: UINT;
	/// Index to actual job in Hashtable
	uintActHastableIdx: UINT;
	///Last new position value from parent
	dinTransportPositionOld_um: DINT;
	///Position correction in faster Task cycletime
	dinPositionCorrection_um: DINT;
	///Difference from actual Tag Position to junction
	dinPositionDifference_um: DINT;
	/// Rising edge of passed sensor
	bolFpPassed: BOOL;
	/// Table Index
	uinWriteTblIndex: UINT;
	/// Hashtable
	aTblDecision: ARRAY[0..cuintMaxIndex] OF T_CheckElement;
	/// Transportposition from last cycle
	dinTransportPositionCalc_old_um: DINT;
	/// Driven Way from last to actual cycle
	dinTransportDifferenz_um: DINT;
	/// Check sensor input cross hanger positv edge
	bolWriteInTableOnce: BOOL;
	/// Blow valve timer
	udiBlowPassingTime_ms: UDINT;
	/// Look for empty hanger position
	dinWaitForEmptyHangerPos_um: DINT;
	/// Look for empty hanger activ
	bolWaitForEmptyHanger: BOOL;
	/// Single, empty hanger generates no signal
	dinPositionWithoutSensorSignal: DINT;
	/// Wait time until jam at slide detected
	udinTimeUntilJamDetected: UDINT;
	/// Star tie for jam at slide
	bolTimeForJamOnce: BOOL;
	/// Open or Close at SUB_WAY1
	bolWay1: BOOL;
	/// Open or Close at SUB_WAY2
	bolWay2: BOOL;
	/// Data ready for writing in table
	bolWriteInTable: BOOL;
	/// Some Vars for Simulation
	bolSetSimuPassedOnce: BOOL;
	/// Positve edge double hanger sensor
	bolDoubleHangerOnce: BOOL;
	/// A Hanger in the table has to be cleared
	bolClearHangerOnce: BOOL;
	/// Positve edge of clearing
	bolClearHanger: BOOL;
	/// Save old position
	dinPositionWithoutSensorSignal_OLD: DINT;
	/// Save postion for detection window
	dinPostionShirtDetected: DINT;
END_VAR
VAR CONSTANT
	///sub States for RELEASE Function
	cSTA_SUB_INITIALIZED: INT := 500;
	cSTA_SUB_WAIT_FOR_JOB: INT := 501;
	///cSTA_SUB_OPEN: INT := 502;
	///cSTA_SUB_CLOSE: INT := 506;
	cSTA_SUB_WAY1: INT := 502;
	cSTA_SUB_WAY2: INT := 506;
	cSTA_SUB_ERROR: INT := 598;
	cSTA_SUB_FINISHED: INT := 600;
END_VAR

(*__________________________________________________________________________________________________
¦	
¦	Vistaprint Schweiz GmbH
¦	CH - 8401 Winterthur
¦
¦	www.vistaprint.ch - info@vistaprint.ch
¦___________________________________________________________________________________________________

Function desription:
Check the hangers and remove the desired 


History:
Version		Date			Author		Comment
---------------------------------------------------------------------------------------------------
0.00.1 		11.10.2013		AVME/MRU	Copied from JUN / DPJ
0.00.2		24.10.2013		AVME/MRU	Some bugs fixed at commissioning
0.00.3		28.10.2013		AVME/MRU	Some changes for different configurations
0.00.4		29.10.2013		AVME/MRU	Some bugs fixed at commissining
0.00.5		30.10.2013		AVME/MRU	Eliminating of compiler warnings
0.00.6		04.11.2013		AVME/MRU	New behavior on error
0.00.7		26.11.2013		VP/RE		Introduced debounce time for double hanger input. Prevents jitter. Btw: Measured signal duration is ~150ms.
0.00.8		16.12.2013		AVME/MRU	in sta_RUN max. pos. reached, neg. pos starts - Bug fixed

___________________________________________________________________________________________________*)


IF (me.bolActivate) THEN // cyclic call enabled
	IF (CIf.Info.bolInitDone=FALSE) THEN // first cycle -> init
		CtrlInit();
		CIf.Info.bolInitDone := TRUE;
	ELSE
		CycleStartDuty();
	
		Always();
		
		StateMachine();
		
		CycleEndDuty();
	END_IF
END_IF;

METHOD PROTECTED Always : BOOL
SUPER^.Always();

// ----------------------------------------------------------------------------------
// cyclic actions outside of statemachine
IF (me.StateMachine.intState<>cSTA_SINGLE_ANSWER) THEN
	SIf.Cur.bolPassed := SIf.In.bolPassed.intern;
	SIf.Cur.bolOpen := SIf.Out.bolOpen.intern;

	; // always error supervision
	
END_IF

// Always change actions in Base Library
// ----------------------------------------------------------------------------------
// overrule error always from base -> no EOFF State!! in EOFF go to OFF
IF (me.StateMachine.intStateNext = cSTA_EOFFBusy) THEN
	IF (me.StateMachine.intState=cSTA_OFF) THEN
		me.StateMachine.intStateNext := cSTA_OFF;
	ELSE // stay in OFF
		me.StateMachine.intStateNext := cSTA_OFFBusy;
	END_IF
END_IF
END_METHOD

METHOD FB_init : BOOL
VAR_INPUT
	///if TRUE, the retain variables are initialized (warm start / cold start)
	bInitRetains: BOOL;
	///if TRUE, the instance afterwards gets moved into the copy code (online change)
	bInCopyCode: BOOL;
END_VAR
VAR
	ii: UINT;
END_VAR
//------------------------------------------------------------------------------------------------------------------------
// to manually change in new FUB implementation!!!
// define valid commands for this controller
FOR ii:= 0 TO (SIZEOF(CIf.Job.aCmdList)/SIZEOF(CIf.Job.aCmdList[0])-1) BY 1 DO
	IF (CIf.Job.aCmdList[ii].intCmd=cCMD_INITIALIZED) THEN
		// found first empty array element
		EXIT;
	END_IF
END_FOR
CIf.Job.aCmdList[ii].intCmd := cCMD_STOP;
CIf.Job.aCmdList[ii].strName := 'Stop'; 
CIf.Job.aCmdList[ii].bolAvailable := TRUE;
ii := ii +1;
CIf.Job.aCmdList[ii].intCmd := cCMD_RUN;
CIf.Job.aCmdList[ii].strName := 'Run'; 
CIf.Job.aCmdList[ii].bolAvailable := TRUE;
ii := ii +1;
CIf.Job.aCmdList[ii].intCmd := cCMD_STOP;
CIf.Job.aCmdList[ii].strName := 'Stop'; 
CIf.Job.aCmdList[ii].bolAvailable := TRUE;
ii := ii +1;

// set name of class/typ
CIf.Info.strType := 'FB_CHD'; 

// set alarm class
SIf.Alm[1].eAlmClass := E_AlmClass.STOP;
SIf.Alm[1].strText := 'timeout passed sensor does not detect the hanger'; 
SIf.Alm[2].eAlmClass := E_AlmClass.INFO;
SIf.Alm[2].strText := 'Cross hanger detection has an hanger rejected';
SIf.Alm[3].eAlmClass := E_AlmClass.STOP;
SIf.Alm[3].strText := 'Open not possible, destination is full';
SIf.Alm[4].eAlmClass := E_AlmClass.TSTOP;
SIf.Alm[4].strText := 'TLP stopped by CHD';


//*******************************************************************************
// initial values
//*******************************************************************************

// software configuration
CIf.SwCfg.bolExist := TRUE;
CIf.SwCfg.bolSimulation := FALSE;

// parmeter
SIf.Par.udiOpenTime_ms := 20;
SIf.Par.udiCloseTime_ms := 10;
SIf.Par.udiPassTime_ms := 10000;
SIf.Par.udiSimPassTime_ms := 500; // SIf.Par.udiPassTime_ms/2;
SIf.Par.dinPosition_um := 10000000;
SIf.Par.dinOpenWay_um := 300000;
SIf.Par.dinDistanceBetweenSensors_DoubleHangerFirst_um := 100000;
SIf.Par.dinDistanceBetweenSensors_EmptyHangerFirst_um := 100000;
SIf.Par.dinPinDistance_um := 305000;
SIf.Par.udinTimeUntilJam_ms := 1000;
SIf.Par.udiPulseLengthBlowValve_ms := 500;
SIf.Par.udiIntervalLengthBlowValve_ms := 10000;
SIf.Par.udiDebounceTimeDoubleHanger_ms := 80;
//*******************************************************************************
// initial values childes
//*******************************************************************************
END_METHOD

METHOD PROTECTED getCmdState : STRING
VAR_INPUT
	intCmdState: INT;
	bolState: BOOL;
END_VAR
getCmdState := SUPER^.getCmdState(intCmdState:=intCmdState,bolState:=bolState); // get global/base defined cmds/states
IF (getCmdState='') THEN // global not defined get local
	// get string cmd/state string information in runtime
	IF (bolState=FALSE) THEN
		// cmd's
(*		CASE intCmdState OF
			; // nothing
		END_CASE;
*)	ELSE
	
	// cmd's
		CASE intCmdState OF
			cSTA_RUNBusy: 
				THIS^.sta_RUNBusy();
			cSTA_RUN: 
				THIS^.sta_RUN();
			cSTA_STOPBusy: 
				THIS^.sta_STOPBusy();
			cSTA_STOP: 
				THIS^.sta_STOP();
				
			// SUB States
			cSTA_SUB_INITIALIZED:
				getCmdState := 'cSTA_SUB_INITIALIZED';
			cSTA_SUB_WAIT_FOR_JOB:
				getCmdState := 'cSTA_SUB_WAIT_FOR_JOB';
(*			cSTA_SUB_OPEN:
				getCmdState := 'cSTA_SUB_OPEN';
			cSTA_SUB_CLOSE:
				getCmdState := 'cSTA_SUB_CLOSE';
*)			cSTA_SUB_WAY1:
				getCmdState := 'cSTA_SUB_WAY1';
			cSTA_SUB_WAY2:
				getCmdState := 'cSTA_SUB_WAY2';
			cSTA_SUB_ERROR:
				getCmdState := 'cSTA_SUB_ERROR';
			cSTA_SUB_FINISHED:
				getCmdState := 'cSTA_SUB_FINISHED';
		END_CASE;
	END_IF
END_IF
END_METHOD

METHOD getCtrlSIf : POINTER TO T_Ctrl_SIf_CHD
getCtrlSIf := ADR(SIf);
END_METHOD

METHOD PROTECTED IoInBridge : BOOL
// digitale and analoge inputs read from hardware or forcing

SIf.In.bolPassed.map := THIS^.In_bolPassed;	// Slide full
SIf.In.bolSensorDoubleHanger.map := THIS^.In_bolDoubleHanger;
SIf.In.bolSensorEmptyHanger.map := THIS^.In_bolEmptyHanger;
SIf.In.bolSensorInconsistentHanger.map := THIS^.In_bolInconsistentHanger;
SIf.In.bolButtonRestartTLP.map := THIS^.In_bolRestartTLP;

IF (CIf.SwCfg.bolSimulation = FALSE) THEN
	
	getInBol(CIf.Job.bolIoForce,ADR(SIf.In.bolPassed));	// Slide full
	
	//getInBol(CIf.Job.bolIoForce,ADR(SIf.In.bolSensorDoubleHanger));
	getInBolDebounced(CIf.Job.bolIoForce, me.FUBInfo.udiSample_ms, Sif.Par.udiDebounceTimeDoubleHanger_ms, ADR(SIf.In.bolSensorDoubleHanger));

	getInBol(CIf.Job.bolIoForce,ADR(SIf.In.bolSensorEmptyHanger));
	getInBol(CIf.Job.bolIoForce,ADR(SIf.In.bolSensorInconsistentHanger));
	getInBol(CIf.Job.bolIoForce,ADR(SIf.In.bolButtonRestartTLP));
ELSE
	//simulation of global IO
END_IF
END_METHOD

METHOD PROTECTED IoOutBridge : BOOL
// digitale and analoge inputs read from hardware or forcing
IF (CIf.SwCfg.bolSimulation = FALSE) THEN
	setOutBol(CIf.Job.bolIoForce ,ADR(SIf.Out.bolOpen));
	setOutBol(CIf.Job.bolIoForce ,ADR(SIf.Out.bolBlow));
	setOutBol(CIf.Job.bolIoForce ,ADR(SIf.Out.bolLightTLPStopedByCHD));
	
	THIS^.Out_bolLightTLPStopedByCHD := SIf.Out.bolLightTLPStopedByCHD.map;
	THIS^.Out_bolOpen := SIf.Out.bolOpen.map;
	THIS^.Out_bolBlow := SIf.Out.bolBlow.map;
END_IF
END_METHOD

METHOD PROTECTED sta_ERROR : BOOL
// state implemetation
//--------------------------------------------------------------------------------------
// Entry action
	IF (me.StateMachine.intState<>me.StateMachine.intStateLastCycle) THEN
		me.StateMachine.intStateHistory := me.StateMachine.intStateLastCycle; // -> possibillity to go back to state before error
		me.StateMachine.intStateLastCycle := me.StateMachine.intState;
		
	END_IF


//--------------------------------------------------------------------------------------
// Cyclic action
	IF (me.StateMachine.intState=me.StateMachine.intStateLastCycle) THEN
		
		IF (SIf.Cfg.bolStopAtRejact) THEN
			;	// Let Junction open
		ELSE
			SIf.Out.bolOpen.intern := 0;
		END_IF
		SIf.Out.bolBlow.intern := 0;
		
		// State Change Condition
		IF 	((CIf.Job.bolAlmReset = TRUE) OR 																// Standart Error Reset
			((Cif.Job.eMe_ActivAlmClass = E_AlmClass.TSTOP) AND SIf.In.bolButtonRestartTLP.intern)) THEN	// Reset CHD with own button
			me.StateMachine.intStateNext := cSTA_ERRORQuit;
		END_IF
	END_IF




//--------------------------------------------------------------------------------------
// Exit action
	IF (me.StateMachine.intState<>me.StateMachine.intStateNext) THEN
		;
	END_IF
END_METHOD

METHOD PROTECTED sta_ERRORQuit : BOOL
// state implemetation
//--------------------------------------------------------------------------------------
// Entry action
	IF (me.StateMachine.intState<>me.StateMachine.intStateLastCycle) THEN
		me.StateMachine.intStateLastCycle := me.StateMachine.intState;
	END_IF


//--------------------------------------------------------------------------------------
// Cyclic action
	IF (me.StateMachine.intState=me.StateMachine.intStateLastCycle) THEN
		
		;
		// evtl. wait time if reset of device is necessary and then decide to go to states or ERROR state
		IF ((CIf.Job.bolAlmReset = TRUE) OR 																// Standart Error Reset
			((Cif.Job.eMe_ActivAlmClass = E_AlmClass.TSTOP) AND SIf.In.bolButtonRestartTLP.intern)) THEN	// Reset CHD with own button
			CIf.Job.eMe_ActivAlmClass := E_AlmClass.NONE; // reset feedback channel for parent
			CIf.Job.bolAlmReset := FALSE;
			SIf.Out.bolOpen.intern := FALSE;	// Reset junction after error
			SIf.Out.bolLightTLPStopedByCHD.intern := FALSE;
		END_IF
		
		// State Change Condition
		IF (CIf.Job.bolAlmReset = FALSE) THEN
			IF (me.StateMachine.intStateHistory<=cSTA_PON) THEN
				me.StateMachine.intStateNext := cSTA_PONBusy;
			ELSIF(me.intCmd=cCMD_OFF) THEN
				me.StateMachine.intStateNext := cSTA_OFFBusy;
			ELSIF(me.intCmd=cCMD_RUN) OR (me.StateMachine.intStateHistory=cSTA_RUN) THEN
				me.StateMachine.intStateNext := cSTA_RUNBusy;
			ELSIF(me.intCmd=cCMD_STOP) THEN
				me.StateMachine.intStateNext := cSTA_STOPBusy;
			END_IF
		END_IF
	END_IF




//--------------------------------------------------------------------------------------
// Exit action
	IF (me.StateMachine.intState<>me.StateMachine.intStateNext) THEN
		;
	END_IF
END_METHOD

METHOD PROTECTED sta_OFF : BOOL
// state implemetation
//--------------------------------------------------------------------------------------
// Entry action
	IF (me.StateMachine.intState<>me.StateMachine.intStateLastCycle) THEN
		me.StateMachine.intStateLastCycle := me.StateMachine.intState;
		
	END_IF


//--------------------------------------------------------------------------------------
// Cyclic action
	IF (me.StateMachine.intState=me.StateMachine.intStateLastCycle) THEN
		
		;
		
		
		// State Change Condition
		IF (me.Alarm.eActivAlmClass<>E_AlmClass.EOFF) AND (me.Alarm.eActivAlmClass<>E_AlmClass.OFF) THEN
			IF (me.intCmd=cCMD_STOP) THEN
				// sensor retract always on cylinder
				me.StateMachine.intStateNext :=  cSTA_STOPBusy;
			ELSIF(me.intCmd=cCMD_RUN) THEN
				me.StateMachine.intStateNext := cSTA_RUNBusy;
			END_IF
		END_IF
	END_IF




//--------------------------------------------------------------------------------------
// Exit action
	IF (me.StateMachine.intState<>me.StateMachine.intStateNext) THEN
		;
	END_IF
END_METHOD

METHOD PROTECTED sta_OFFBusy : BOOL
// state implemetation
//--------------------------------------------------------------------------------------
// Entry action
	IF (me.StateMachine.intState<>me.StateMachine.intStateLastCycle) THEN
		me.StateMachine.intStateLastCycle := me.StateMachine.intState;
		
	END_IF


//--------------------------------------------------------------------------------------
// Cyclic action
	IF (me.StateMachine.intState=me.StateMachine.intStateLastCycle) THEN
		
		// switch VALVE off
		SIf.Out.bolOpen.intern := FALSE;
		SIf.Out.bolBlow.intern := FALSE;
		
		
		
		// State Change Condition
		IF (FALSE) THEN
			;
		ELSIF (TRUE) THEN
			me.StateMachine.intStateNext := cSTA_OFF;
		END_IF
	END_IF




//--------------------------------------------------------------------------------------
// Exit action
	IF (me.StateMachine.intState<>me.StateMachine.intStateNext) THEN
		;
	END_IF
END_METHOD

METHOD PROTECTED sta_PON : BOOL
// state implemetation
//--------------------------------------------------------------------------------------
// Entry action
	IF (me.StateMachine.intState<>me.StateMachine.intStateLastCycle) THEN
		me.StateMachine.intStateLastCycle := me.StateMachine.intState;
		
	END_IF


//--------------------------------------------------------------------------------------
// Cyclic action
	IF (me.StateMachine.intState=me.StateMachine.intStateLastCycle) THEN
		
		;
		
		
		// State Change Condition
		IF(me.intCmd=cCMD_OFF) THEN
			me.StateMachine.intStateNext := cSTA_OFFBusy;
		ELSIF(me.intCmd=cCMD_RUN) THEN
			me.StateMachine.intStateNext := cSTA_OFFBusy;
		ELSIF(me.intCmd=cCMD_STOP) THEN
			me.StateMachine.intStateNext := cSTA_STOPBusy;
		END_IF
	END_IF




//--------------------------------------------------------------------------------------
// Exit action
	IF (me.StateMachine.intState<>me.StateMachine.intStateNext) THEN
		;
	END_IF
END_METHOD

METHOD PROTECTED sta_RUN : BOOL
// state implemetation
//--------------------------------------------------------------------------------------
// Entry action
	IF (me.StateMachine.intState<>me.StateMachine.intStateLastCycle) THEN
		me.StateMachine.intStateLastCycle := me.StateMachine.intState;
			
		me.SubStateMachine.intState := cSTA_SUB_WAIT_FOR_JOB; // init sub state machine
		me.SubStateMachine.intStateNext := cSTA_SUB_WAIT_FOR_JOB; // init sub state machine
		fbSimulationTimer.PT := UDINT_TO_TIME(SIf.Par.udiSimPassTime_ms);
		fbSimulationTimer(); // set time/reset timer

	END_IF


//--------------------------------------------------------------------------------------
// Cyclic action
	IF (me.StateMachine.intState=me.StateMachine.intStateLastCycle) THEN
		// Simulation
		IF (CIf.SwCfg.bolSimulation) THEN
			fbSimulationTimer(); // set time/reset timer
			IF (SIf.Out.bolOpen.intern = TRUE) THEN 
				fbSimulationTimer.IN := TRUE;
			ELSIF (SIf.Out.bolOpen.intern = FALSE) AND (fbSimulationTimer.Q = TRUE) THEN
				fbSimulationTimer.IN := FALSE;			
			END_IF
			IF (fbSimulationTimer.Q = TRUE) AND (bolSetSimuPassedOnce = FALSE) THEN
				SIf.In.bolPassed.intern := TRUE;
				bolSetSimuPassedOnce := TRUE;
			ELSE
				SIf.In.bolPassed.intern := FALSE;
			END_IF
			IF (fbSimulationTimer.Q = FALSE) THEN
				bolSetSimuPassedOnce := FALSE;	
			END_IF
		END_IF
		
		//--------------------------------------------------------------------------------------
		// Always RUN actions
		
		// If this task is in faster cycle then the parent, calculate internal position more exactly during the taskcycle
		IF dinTransportPositionOld_um <> SIf.Cur.dinTransportPosition_um THEN
			SIf.Cur.dinTransportPositionCalc_um := SIf.Cur.dinTransportPosition_um;
			dinTransportPositionOld_um := SIf.Cur.dinTransportPosition_um;
			dinPositionCorrection_um := 0;
		ELSE
			dinPositionCorrection_um := dinPositionCorrection_um + LREAL_TO_DINT(DINT_TO_LREAL(SIf.Cur.dinTransportspeed_um_s) * UDINT_TO_LREAL(me.FUBInfo.udiSample_ms) / 1000.0 );
			SIf.Cur.dinTransportPositionCalc_um := dinTransportPositionOld_um + dinPositionCorrection_um;
		END_IF
		
		// Check for double hanger (Sensors: just double hanger, if nothing seen -> junction closed)
		// -> Write bad hangers to table
		IF (SIf.Cfg.bolHasEmptyHangerSensor = FALSE) THEN
			IF (SIf.In.bolSensorDoubleHanger.intern = TRUE) THEN
				bolWriteInTable := TRUE;
			ELSE
				bolWriteInTable := FALSE;
				bolWriteInTableOnce := FALSE;
			END_IF
			bolWay1 := TRUE;	// WAY1 = OPEN
			bolWay2 := FALSE;	// WAY2 = CLOSE
		// Check for double hanger (Sensors: Double hanger, empty hanger, if nothing seen -> junction open)
		// -> Write good hangers to table
		ELSE
			IF ((SIf.In.bolSensorDoubleHanger.intern = TRUE) AND (bolWaitForEmptyHanger = FALSE)) THEN
				dinWaitForEmptyHangerPos_um := SIf.Cur.dinTransportPositionCalc_um + SIf.Par.dinDistanceBetweenSensors_DoubleHangerFirst_um;
				bolWaitForEmptyHanger := TRUE;
				// DoubleHanger comes to late, Hanger already in table -> clear is needed
				IF (bolWriteInTable AND (bolClearHanger= FALSE)) THEN
					bolClearHanger := TRUE;
				END_IF	
			ELSE
				bolClearHanger := FALSE;
				bolClearHangerOnce := FALSE;
			END_IF
			
			IF (bolWaitForEmptyHanger = TRUE) THEN	// DoubleHanger detected -> doesn't care with or without shirt
				IF (dinWaitForEmptyHangerPos_um < SIf.Cur.dinTransportPositionCalc_um) THEN // Empty Hanger, write in Table
					bolWaitForEmptyHanger := FALSE;
				END_IF
			ELSE // No DoubleHanger detected -> if Not EmptyHanger then it is a valid Hanger
				IF ((SIf.In.bolSensorEmptyHanger.intern = TRUE) AND (bolWriteInTableOnce = FALSE)) THEN	
					bolWriteInTable := TRUE;
					dinPostionShirtDetected := SIf.Cur.dinTransportPositionCalc_um;
//				ELSIF (SIf.In.bolSensorEmptyHanger.intern = FALSE) THEN
				ELSIF ((SIf.In.bolSensorEmptyHanger.intern = FALSE) AND (SIf.Cur.dinTransportPositionCalc_um > (dinPostionShirtDetected+SIf.Par.dinDistanceBetweenSensors_EmptyHangerFirst_um))) THEN
					bolWriteInTableOnce := FALSE;
					bolWriteInTable := FALSE;
				// Max dint value reached, position starts with max negativ position
				ELSIF ((dinPostionShirtDetected >0 ) AND (SIf.Cur.dinTransportPositionCalc_um < 0) AND (SIf.In.bolSensorEmptyHanger.intern = FALSE)) THEN
					bolWriteInTableOnce := FALSE;
					bolWriteInTable := FALSE;
				END_IF
			END_IF
			bolWay1 := FALSE;	// WAY1 = OPEN
			bolWay2 := TRUE;	// WAY2 = CLOSE
		END_IF
		
		// Write in table
		IF	((bolWriteInTable = TRUE) AND (bolWriteInTableOnce = FALSE)) THEN
			uinWriteTblIndex := uinWriteTblIndex + 1;
			IF uinWriteTblIndex > cuintMaxIndex THEN
				uinWriteTblIndex := 0;
			END_IF
			dinPositionWithoutSensorSignal_OLD:= dinPositionWithoutSensorSignal;	// Save Old Position
			bolWriteInTableOnce:= TRUE;
			aTblDecision[uinWriteTblIndex].eState := E_DecisionState.WayToJunction;
			aTblDecision[uinWriteTblIndex].dinActPos_um := 1;	
		END_IF
		IF (bolClearHanger AND NOT bolClearHangerOnce) THEN // Clear HangerHasShirt if a DoubleHanger is detected
			bolClearHangerOnce:= TRUE;						// Do it Once
			aTblDecision[uinWriteTblIndex].eState := E_DecisionState.Processed;	// Nothing to Do
			aTblDecision[uinWriteTblIndex].dinActPos_um := -1;					// No Position needed
			dinPositionWithoutSensorSignal:= dinPositionWithoutSensorSignal_OLD;// Restore old Position
		END_IF
		
		// Increase the position of every Hanger in the table, if it is on the way to junction
		dinTransportDifferenz_um := SIf.Cur.dinTransportPositionCalc_um - dinTransportPositionCalc_old_um;
		FOR uinI := 0 TO cuintMaxIndex DO
			IF ((aTblDecision[uinI].eState = E_DecisionState.WayToJunction) OR (aTblDecision[uinI].eState = E_DecisionState.OnJunction)) THEN
				aTblDecision[uinI].dinActPos_um := aTblDecision[uinI].dinActPos_um + dinTransportDifferenz_um;
			END_IF
		END_FOR	
		dinTransportPositionCalc_old_um := SIf.Cur.dinTransportPositionCalc_um;
		
		// Check table if there is a job
		dinPositionDifference_um := SIf.Par.dinPosition_um; // Set maximal value to search the smalles one
		// Loop through the table
		FOR uinI := 0 TO cuintMaxIndex DO
			// Check if this job is on the way to the junction
			IF aTblDecision[uinI].eState = E_DecisionState.WayToJunction THEN
				// Chech if it is the nearest tag
				IF 	dinPositionDifference_um > SIf.Par.dinPosition_um - aTblDecision[uinI].dinActPos_um THEN
					dinPositionDifference_um := SIf.Par.dinPosition_um - aTblDecision[uinI].dinActPos_um;
					uintNextHastableIdx := uinI;
				END_IF
			END_IF
		END_FOR
		IF ((dinPositionDifference_um = SIf.Par.dinPosition_um) OR 			// No Hanger found
			(dinPositionDifference_um > SIf.Par.dinPinDistance_um)) THEN 	// Pin without information is nearest
			dinPositionWithoutSensorSignal:= dinPositionWithoutSensorSignal + dinTransportDifferenz_um;
		ELSE
			dinPositionWithoutSensorSignal:= 0;								// Good hanger on way to junction
		END_IF
		
		// A hanger is on slide message
		IF ((SIf.In.bolPassed.intern = TRUE) AND (bolFpPassed = FALSE)) THEN
			bolFpPassed := TRUE;
			udinTimeUntilJamDetected:= 0;
				
			IF SIf.cfg.bolStopAtRejact THEN
				IF (SIf.Cfg.bolHasEmptyHangerSensor = TRUE) THEN // Just if Emty Hanger Exist
					// Set Alarm: SIf.Alm[4].strText := 'TLP stopped by CHD';
					pfbAlarmCtrl^.setAlarm(CIf.Info.intCtrlId,4,0,ADR(SIf.Alm),E_AlmState.RST,CIf.Job.eMe_ActivAlmClass);
					me.SubStateMachine.intStateNext := cSTA_SUB_ERROR;
					SIf.Out.bolLightTLPStopedByCHD.intern := TRUE;
				END_IF
				; //Else No message needed
			ELSE	
				// Set Alarm: SIf.Alm[2].strText := 'Cross hanger detection has an hanger rejected';
				pfbAlarmCtrl^.setAlarm(CIf.Info.intCtrlId,2,0,ADR(SIf.Alm),E_AlmState.RST,CIf.Job.eMe_ActivAlmClass);	
			END_IF
		ELSIF (SIf.In.bolPassed.intern = FALSE) THEN
			bolFpPassed := FALSE;
		END_IF
		// Jam on slide message
		IF (bolFpPassed = TRUE) THEN
			udinTimeUntilJamDetected:= udinTimeUntilJamDetected + me.FUBInfo.udiSample_ms;
			IF (udinTimeUntilJamDetected > SIf.Par.udinTimeUntilJam_ms) THEN
				// SIf.Alm[3].strText := 'Open not possible, destination is full';
				pfbAlarmCtrl^.setAlarm(CIf.Info.intCtrlId,3,0,ADR(SIf.Alm),E_AlmState.RST,CIf.Job.eMe_ActivAlmClass);
			END_IF
		END_IF

		
		// Count double hanger
		IF (SIf.In.bolSensorDoubleHanger.intern AND NOT bolDoubleHangerOnce) THEN
			SIf.Cur.udintCounterDoubleHanger := SIf.Cur.udintCounterDoubleHanger + 1;
			bolDoubleHangerOnce := TRUE;
		ELSIF (SIf.In.bolSensorDoubleHanger.intern = FALSE) THEN
			bolDoubleHangerOnce := FALSE;
		END_IF
		
		//--------------------------------------------------------------------------------------
		// sub state machine for sequence
		CASE me.SubStateMachine.intState OF
			//--------------------------------------------------------------------------------------
			cSTA_SUB_WAIT_FOR_JOB:
				IF (me.SubStateMachine.intState<>me.SubStateMachine.intStateLastCycle) THEN
					me.SubStateMachine.intStateLastCycle := me.SubStateMachine.intState;
				END_IF
				// State Change Condition
				// Simulation
				IF (CIf.SwCfg.bolSimulation) THEN
					;// SIf.In.bolPassed.intern := FALSE;
				END_IF
				
				
				// If reaction way (time*speed) is bigger then the rest of the way to the junction, close
				IF dinPositionDifference_um <= LREAL_TO_DINT( UDINT_TO_LREAL(SIf.Par.udiCloseTime_ms) * DINT_TO_LREAL(SIf.Cur.dinTransportspeed_um_s) ) / 1000.0 THEN
					me.SubStateMachine.intStateNext := cSTA_SUB_WAY1;	// cSTA_SUB_CLOSE;
				// Empty hanger or crossed hanger at (junction - reaction way)
				ELSIF (dinPositionWithoutSensorSignal >= (SIf.Par.dinPinDistance_um - LREAL_TO_DINT( UDINT_TO_LREAL(SIf.Par.udiOpenTime_ms) * DINT_TO_LREAL(SIf.Cur.dinTransportspeed_um_s))/1000.0)) THEN
//					IF (SIf.In.bolPassed.intern = FALSE) THEN
						me.SubStateMachine.intStateNext := cSTA_SUB_WAY2;	// cSTA_SUB_OPEN;
//						bolTimeForJamOnce := FALSE;	
//					ELSE
(*						IF (bolTimeForJamOnce = FALSE) THEN
							udinTimeUntilJamDetected:= me.StateMachine.udiTimeInState_ms + SIf.Par.udinTimeUntilJam_ms;
							bolTimeForJamOnce := TRUE;	
						END_IF
						IF (bolTimeForJamOnce AND (udinTimeUntilJamDetected < me.StateMachine.udiTimeInState_ms)) THEN
*)							// SIf.Alm[3].strText := 'Open not possible, destination is full';
//							pfbAlarmCtrl^.setAlarm(CIf.Info.intCtrlId,3,0,ADR(SIf.Alm),E_AlmState.RST,CIf.Job.eMe_ActivAlmClass);
//							me.SubStateMachine.intStateNext := cSTA_SUB_WAY2;
(*							me.SubStateMachine.intStateNext := cSTA_sub_ERROR;
							bolTimeForJamOnce := FALSE;
						END_IF
*)//				END_IF
				END_IF

			//--------------------------------------------------------------------------------------
			cSTA_SUB_WAY1: //CLOSE
				IF (me.SubStateMachine.intState<>me.SubStateMachine.intStateLastCycle) THEN
					me.SubStateMachine.intStateLastCycle := me.SubStateMachine.intState;

					uintActHastableIdx := uintNextHastableIdx;
					aTblDecision[uintNextHastableIdx].eState := E_DecisionState.OnJunction;
					
				END_IF
					
				SIf.Out.bolOpen.intern := bolWay1;	// FALSE
					
				// Simulation
				IF (CIf.SwCfg.bolSimulation) THEN
					;
				END_IF
					
				// Check position
				IF (SIf.Par.dinPosition_um + SIf.Par.dinOpenWay_um <= aTblDecision[uintActHastableIdx].dinActPos_um + dinPositionCorrection_um) THEN
					IF aTblDecision[uintActHastableIdx].eState < E_DecisionState.Processed THEN
						// Only set to processe if not allready driven out
						aTblDecision[uintActHastableIdx].eState := E_DecisionState.Processed;
					END_IF					
					aTblDecision[uintActHastableIdx].dinActPos_um := -2;
				END_IF
					
				// State Change Condition
				// Check error if tray never reach the output
				IF (me.SubStateMachine.udiTimeInState_ms > SIf.Par.udiPassTime_ms) THEN
					// Set Alarm: SIf.Alm[1].strText := 'timeout passed sensor does not detect the hanger'; 
					pfbAlarmCtrl^.setAlarm(CIf.Info.intCtrlId,1,0,ADR(SIf.Alm),E_AlmState.RST,CIf.Job.eMe_ActivAlmClass);
					me.SubStateMachine.intStateNext := cSTA_SUB_ERROR;
				// Check if tray allready passed
			//	ELSIF (aTblDecision[intActHastableIdx].eState > E_DecisionState.OnJunction) AND (dinPositionDifference_um < LREAL_TO_DINT ( UDINT_TO_LREAL(SIf.Par.udiCloseTime_ms) * DINT_TO_LREAL(SIf.Cur.dinTransportspeed_um_s) / 1000.0 ) ) THEN
			//		me.SubStateMachine.intStateNext := cSTA_SUB_WAY1;	// cSTA_SUB_CLOSE;
				ELSIF (aTblDecision[uintActHastableIdx].eState > E_DecisionState.OnJunction) THEN	
					IF (SIf.cfg.bolStopAtRejact AND (SIf.Cfg.bolHasEmptyHangerSensor = FALSE)) THEN // Just if no Emty Hanger Exist
						// Set Alarm: SIf.Alm[4].strText := 'TLP stopped by CHD';
						pfbAlarmCtrl^.setAlarm(CIf.Info.intCtrlId,4,0,ADR(SIf.Alm),E_AlmState.RST,CIf.Job.eMe_ActivAlmClass);
						me.SubStateMachine.intStateNext := cSTA_SUB_ERROR;
						SIf.Out.bolLightTLPStopedByCHD.intern := TRUE;
					ELSE
						me.SubStateMachine.intStateNext := cSTA_SUB_WAIT_FOR_JOB;
					END_IF
				END_IF

			//--------------------------------------------------------------------------------------
			cSTA_SUB_WAY2:	// OPEN:
				IF (me.SubStateMachine.intState<>me.SubStateMachine.intStateLastCycle) THEN
					me.SubStateMachine.intStateLastCycle := me.SubStateMachine.intState;
				END_IF
				
				SIf.Out.bolOpen.intern := bolWay2;	// TRUE;
					
				// Simulation
					
					
				// State Change Condition
				me.SubStateMachine.intStateNext := cSTA_SUB_WAIT_FOR_JOB;
				dinPositionWithoutSensorSignal := 0;

				// Simulation
				IF (CIf.SwCfg.bolSimulation) THEN
					;// SIf.In.bolPassed.intern := FALSE;
				END_IF
				
			//--------------------------------------------------------------------------------------
			cSTA_SUB_ERROR:
				IF (me.SubStateMachine.intState<>me.SubStateMachine.intStateLastCycle) THEN
					me.SubStateMachine.intStateLastCycle := me.SubStateMachine.intState;
				END_IF
				
				IF (SIf.cfg.bolStopAtRejact) THEN 
					;	// Let Junction open
				ELSE
					SIf.Out.bolOpen.intern := FALSE;
				END_IF
				
				// State Change Condition
				// No change, going over an other main state
					
		END_CASE
		
		// ------------------------------------------------------
		// Blow valve
		IF (udiBlowPassingTime_ms > Sif.par.udiIntervalLengthBlowValve_ms) THEN
			IF (udiBlowPassingTime_ms > (SIf.Par.udiIntervalLengthBlowValve_ms + SIf.Par.udiPulseLengthBlowValve_ms)) THEN
				SIf.Out.bolBlow.intern := FALSE;
				udiBlowPassingTime_ms := 0;
			ELSE
				SIf.Out.bolBlow.intern := TRUE;
			END_IF
		END_IF
				
		udiBlowPassingTime_ms := udiBlowPassingTime_ms + me.FUBInfo.udiSample_ms;
		// ------------------------------------------------------
		
		// State Change Condition
		// Check error if retracted position not reached
		IF me.SubStateMachine.intState = cSTA_SUB_ERROR THEN
			me.StateMachine.intStateNext :=  cSTA_ERROR;
		ELSIF(me.intCmd=cCMD_STOP) THEN
			me.StateMachine.intStateNext := cSTA_STOPBusy;
		END_IF
	END_IF




//--------------------------------------------------------------------------------------
// Exit action
	IF (me.StateMachine.intState<>me.StateMachine.intStateNext) THEN
		;
	END_IF
END_METHOD

METHOD PROTECTED sta_RUNBusy : BOOL
// state implemetation
//--------------------------------------------------------------------------------------
// Entry action
	IF (me.StateMachine.intState<>me.StateMachine.intStateLastCycle) THEN
		me.StateMachine.intStateLastCycle := me.StateMachine.intState;
					
	END_IF


//--------------------------------------------------------------------------------------
// Cyclic action
	IF (me.StateMachine.intState=me.StateMachine.intStateLastCycle) THEN
	
	
		FOR uinWriteTblIndex := 0 TO cuintMaxIndex DO	// Clear table before RUN
			aTblDecision[uinWriteTblIndex].eState := E_DecisionState.none;
			aTblDecision[uinWriteTblIndex].dinActPos_um := 0;
		END_FOR	
		uinWriteTblIndex := 0;
				
		
		// State Change Condition
		me.StateMachine.intStateNext := cSTA_RUN;		
	END_IF
	



//--------------------------------------------------------------------------------------
// Exit action
	IF (me.StateMachine.intState<>me.StateMachine.intStateNext) THEN
		;
	END_IF
END_METHOD

METHOD PROTECTED sta_STOP : BOOL
// state implemetation
//--------------------------------------------------------------------------------------
// Entry action
	IF (me.StateMachine.intState<>me.StateMachine.intStateLastCycle) THEN
		me.StateMachine.intStateLastCycle := me.StateMachine.intState;
		
	END_IF


//--------------------------------------------------------------------------------------
// Cyclic action
	IF (me.StateMachine.intState=me.StateMachine.intStateLastCycle) THEN
	
		
		// State Change Condition
		IF (me.intCmd=cCMD_RUN) THEN
			me.StateMachine.intStateNext := cSTA_RUNBusy;
		END_IF
	END_IF




//--------------------------------------------------------------------------------------
// Exit action
	IF (me.StateMachine.intState<>me.StateMachine.intStateNext) THEN
		;
	END_IF
END_METHOD

METHOD PROTECTED sta_STOPBusy : BOOL
// state implemetation
//--------------------------------------------------------------------------------------
// Entry action
	IF (me.StateMachine.intState<>me.StateMachine.intStateLastCycle) THEN
		me.StateMachine.intStateLastCycle := me.StateMachine.intState;

	END_IF


//--------------------------------------------------------------------------------------
// Cyclic action
	IF (me.StateMachine.intState=me.StateMachine.intStateLastCycle) THEN

		// Simulation
		
		//no change action
		SIf.Out.bolOpen.intern := FALSE;
		SIf.Out.bolBlow.intern := FALSE;
		
		// State Change Condition
		IF (me.StateMachine.udiTimeInState_ms > SIf.Par.udiCloseTime_ms) THEN
			me.StateMachine.intStateNext := cSTA_STOP;
		END_IF
	END_IF




//--------------------------------------------------------------------------------------
// Exit action
	IF (me.StateMachine.intState<>me.StateMachine.intStateNext) THEN
		;
	END_IF
END_METHOD

METHOD PROTECTED StateMachine : BOOL
SUPER^.StateMachine();

// main statemachine of base controller
CASE me.StateMachine.intState OF
    cSTA_RUNBusy: 
        THIS^.sta_RUNBusy();
    cSTA_RUN: 
        THIS^.sta_RUN();
     cSTA_STOPBusy: 
        THIS^.sta_STOPBusy();
    cSTA_STOP: 
        THIS^.sta_STOP();
END_CASE;
END_METHOD

END_FUNCTION_BLOCK

// POUs/Controller/Lvl0/FOC (Folder Communication)/FB_FOC
FUNCTION_BLOCK FB_FOC EXTENDS FB_CtrlBase
VAR_INPUT
	/// 0=No Error
	In_usiCANDeviceErrorState: USINT;
END_VAR
VAR
	fbReceiveFolderState: FB_ReceiveFolderState;
	fbSendFolderMessage: FB_SendFolderMessage;
	/// interface to LineControl
	bolSEND_CAN_MESSAGE: BOOL;
	bolCanMessageOk: BOOL;
	bolOldSendCanMessage: BOOL;
	/// Specific interface struct for public access
	SIf: T_Ctrl_SIf_FOC;
	/// current counter flag
	uliOldSentMessagesCount: ULINT;
	/// current counter
	uliSentMessagesCount: ULINT;
	bolOldFilteredDataReadReady: BOOL;
	bolOldFilteredEmptyHanger: BOOL;
	tSendMessageTimer: TON;
	udiTimeSinceLastCanMessage: UDINT;
	udiTimeSinceLastDataReadReadyTrue: UDINT;
	udiTimeSinceLastDataReadReadyFalse: UDINT;
	bolSendMessage: BOOL;
	bolReleaseShirtsRequested: BOOL;
END_VAR

